// POUs/Local/Objects/FB_BACnet_AV_Disp
// Analog Setpoint Object for Operation
// - Used to display a value
{attribute 'enable_dynamic_creation'}
FUNCTION_BLOCK FB_BACnet_AV_Disp EXTENDS FB_BACnet_Object
VAR_INPUT
	fVal			: REAL;
END_VAR
VAR_INPUT CONSTANT PERSISTENT
	{region 'Variable Parameters'}
		{attribute 'parameterCategory':='Value'}
		fCOVIncrement : REAL := 0.1;
		{attribute 'parameterCategory':='Value'}
		eUnit : E_BA_Unit := E_BA_Unit.eOther_NoUnits;
	{endregion}
END_VAR
VAR_OUTPUT
	fPresVal	: REAL;
END_VAR

IF bReady THEN
	fPresVal := fVal;
ELSE
	fPresVal := 0;
END_IF

SUPER^();

METHOD PROTECTED OnObjectStateChanged
SUPER^.OnObjectStateChanged();

CASE (tState) OF
	TCOM_STATE.TCOM_STATE_PREOP:
		// SyncHandler:
		RequestSyncHandlers(2, 3);
		
		// Properties:
		// EnableProperty(E_BACnetPropIdentifier.PropDeviceType, FALSE);
		EnableProperty(E_BACnetPropIdentifier.PropNotificationClass, FALSE);
		EnableProperty(E_BACnetPropIdentifier.PropNotifyType, FALSE);
		EnableProperty(E_BACnetPropIdentifier.PropEventEnable, FALSE);
		EnableProperty(E_BACnetPropIdentifier.PropEventTimeStamps, FALSE);
		EnableProperty(E_BACnetPropIdentifier.PropEventMessageTexts, FALSE);
		EnableProperty(E_BACnetPropIdentifier.PropEventMessageTextsConfig, FALSE);
		EnableProperty(E_BACnetPropIdentifier.PropTimeDelay, FALSE);
		EnableProperty(E_BACnetPropIdentifier.PropAckedTransitions, FALSE);
		EnableProperty(E_BACnetPropIdentifier.PropReliability, FALSE);
		EnableProperty(E_BACnetPropIdentifier.PropEventDetectionEnable, FALSE);
		EnableProperty(E_BACnetPropIdentifier.PropEventAlgorithmInhibit, FALSE);
		EnableProperty(E_BACnetPropIdentifier.PropTimeDelayNormal, FALSE);
		EnableProperty(E_BACnetPropIdentifier.PropReliabilityEvaluationInhibit, FALSE);
		EnableProperty(E_BACnetPropIdentifier.PropLimitEnable, FALSE);
		EnableProperty(E_BACnetPropIdentifier.PropHighLimit, FALSE);
		EnableProperty(E_BACnetPropIdentifier.PropLowLimit, FALSE);
		EnableProperty(E_BACnetPropIdentifier.PropDeadband, FALSE);
		EnableProperty(E_BACnetPropIdentifier.PropRelinquishDefault, FALSE);
		EnableProperty(E_BACnetPropIdentifier.PropPriorityArray, FALSE);
		EnableProperty(E_BACnetPropIdentifier.PropCurrentlyActivePriority, FALSE);
		
		WriteProtectProperty(E_BACnetPropIdentifier.PropOutOfService, TRUE);
		// EnableProperty(E_BACnetPropIdentifier.PropStatusFlags, FALSE);
		// EnableProperty(E_BACnetPropIdentifier.PropEventState, FALSE);
		
		WriteProtectProperty(E_BACnetPropIdentifier.PropPresentValue, TRUE);

	TCOM_STATE.TCOM_STATE_SAFEOP:
		SyncProperty(E_BACnetPropIdentifier.PropPresentValue, SIZEOF(fVal), ADR(fVal), 0, eSync_ToSupplement);	
	
	TCOM_STATE.TCOM_STATE_OP:
		SyncProperty(E_BACnetPropIdentifier.PropUnits, SIZEOF(eUnit), ADR(eUnit), 0, eFullSync_InitPLC);
		SyncProperty(E_BACnetPropIdentifier.PropCovIncrement, SIZEOF(fCOVIncrement), ADR(fCOVIncrement), 0, eFullSync_InitPLC);
		
END_CASE
END_METHOD

METHOD FB_init : BOOL
VAR_INPUT
	bInitRetains : BOOL; // if TRUE, the retain variables are initialized (warm start / cold start)
	bInCopyCode : BOOL;  // if TRUE, the instance afterwards gets moved into the copy code (online change)
END_VAR
eObjectType := E_BACnetObjType.ObjAnalogValue;
END_METHOD

END_FUNCTION_BLOCK

// POUs/Local/Objects/FB_BACnet_AV_Setp
// Analog Setpoint Object for Operation
// - Used to define a setpoint by user
{attribute 'enable_dynamic_creation'}
FUNCTION_BLOCK FB_BACnet_AV_Setp EXTENDS FB_BACnet_Object
VAR_INPUT CONSTANT PERSISTENT
	{region 'Variable Parameters'}
		{attribute 'parameterCategory':='Value'}
		fCOVIncrement : REAL := 0.1;
		{attribute 'parameterCategory':='Value'}
		eUnit : E_BA_Unit := E_BA_Unit.eOther_NoUnits;
	{endregion}
	{region 'Operational Parameters'}
		{attribute 'parameterCategory':='Value'}
		fValue : REAL;
	{endregion}
END_VAR
VAR_OUTPUT
	fPresVal	: REAL;
END_VAR

IF bReady THEN
	fPresVal := fValue;
ELSE
	fPresVal := 0;
END_IF

SUPER^();

METHOD PROTECTED OnObjectStateChanged
SUPER^.OnObjectStateChanged();

CASE (tState) OF
	TCOM_STATE.TCOM_STATE_PREOP:
		// SyncHandler:
		RequestSyncHandlers(3, 3);
		
		// Properties:
		// DisableProperty(E_BACnetPropIdentifier.PropDeviceType, FALSE);
		EnableProperty(E_BACnetPropIdentifier.PropNotificationClass, FALSE);
		EnableProperty(E_BACnetPropIdentifier.PropNotifyType, FALSE);
		EnableProperty(E_BACnetPropIdentifier.PropEventEnable, FALSE);
		EnableProperty(E_BACnetPropIdentifier.PropEventTimeStamps, FALSE);
		EnableProperty(E_BACnetPropIdentifier.PropEventMessageTexts, FALSE);
		EnableProperty(E_BACnetPropIdentifier.PropEventMessageTextsConfig, FALSE);
		EnableProperty(E_BACnetPropIdentifier.PropTimeDelay, FALSE);
		EnableProperty(E_BACnetPropIdentifier.PropAckedTransitions, FALSE);
		EnableProperty(E_BACnetPropIdentifier.PropReliability, FALSE);
		EnableProperty(E_BACnetPropIdentifier.PropEventDetectionEnable, FALSE);
		EnableProperty(E_BACnetPropIdentifier.PropEventAlgorithmInhibit, FALSE);
		EnableProperty(E_BACnetPropIdentifier.PropTimeDelayNormal, FALSE);
		EnableProperty(E_BACnetPropIdentifier.PropReliabilityEvaluationInhibit, FALSE);
		EnableProperty(E_BACnetPropIdentifier.PropLimitEnable, FALSE);
		EnableProperty(E_BACnetPropIdentifier.PropHighLimit, FALSE);
		EnableProperty(E_BACnetPropIdentifier.PropLowLimit, FALSE);
		EnableProperty(E_BACnetPropIdentifier.PropDeadband, FALSE);
		EnableProperty(E_BACnetPropIdentifier.PropRelinquishDefault, FALSE);
		EnableProperty(E_BACnetPropIdentifier.PropPriorityArray, FALSE);
		EnableProperty(E_BACnetPropIdentifier.PropCurrentlyActivePriority, FALSE);
		
		WriteProtectProperty(E_BACnetPropIdentifier.PropOutOfService, TRUE);
		// EnableProperty(E_BACnetPropIdentifier.PropStatusFlags, FALSE);
		// EnableProperty(E_BACnetPropIdentifier.PropEventState, FALSE);
		
	TCOM_STATE.TCOM_STATE_SAFEOP:
		;
		
	TCOM_STATE.TCOM_STATE_OP:
		SyncProperty(E_BACnetPropIdentifier.PropPresentValue, SIZEOF(fValue), ADR(fValue), 0, eFullSync_InitPLC);
		
		SyncProperty(E_BACnetPropIdentifier.PropUnits, SIZEOF(eUnit), ADR(eUnit), 0, eFullSync_InitPLC);
		SyncProperty(E_BACnetPropIdentifier.PropCovIncrement, SIZEOF(fCOVIncrement), ADR(fCOVIncrement), 0, eFullSync_InitPLC);
		
END_CASE
END_METHOD

METHOD FB_init : BOOL
VAR_INPUT
	bInitRetains : BOOL; // if TRUE, the retain variables are initialized (warm start / cold start)
	bInCopyCode : BOOL;  // if TRUE, the instance afterwards gets moved into the copy code (online change)
END_VAR
eObjectType := E_BACnetObjType.ObjAnalogValue;
END_METHOD

END_FUNCTION_BLOCK

// POUs/Local/Objects/FB_BACnet_BI_Raw
// Binary Input Object
// - Raw communication
{attribute 'pin_presentation_order_outputs' := 'bPresVal,bEvent,eRlbty'}
{attribute 'enable_dynamic_creation'}
FUNCTION_BLOCK FB_BACnet_BI_Raw EXTENDS FB_BACnet_BaseBI
VAR_INPUT
	bRawVal					: BOOL;				// Raw value
END_VAR
VAR_INPUT CONSTANT PERSISTENT
	{region 'Fixed Parameters'}
		{attribute 'parameterCategory':='Hardware'}
		nIoBusNr : BYTE := 16#FF;
	{endregion}
END_VAR

SUPER^();

METHOD PROTECTED OnObjectStateChanged
SUPER^.OnObjectStateChanged();

CASE (tState) OF
	TCOM_STATE.TCOM_STATE_PREOP:
		// SyncHandler:
		RequestSyncHandlers(0, 1);

		IF (nIoBusNr <> 16#FF) THEN
			WritePropertyByte(E_BACnetPropIdentifier.PropIoBusNr, nIoBusNr);
		END_IF
		
	TCOM_STATE.TCOM_STATE_SAFEOP:
		SyncProperty(E_BACnetPropIdentifier.PropRawIoBinaryValueBOOL, SIZEOF(bRawVal), ADR(bRawVal), 0, eSync_ToSupplement);
		
	TCOM_STATE.TCOM_STATE_OP:
		;
		
END_CASE
END_METHOD

END_FUNCTION_BLOCK

// POUs/Local/Objects/[Base]/FB_BACnet_BaseBI
FUNCTION_BLOCK ABSTRACT FB_BACnet_BaseBI EXTENDS FB_BACnet_EventObject
VAR_INPUT CONSTANT PERSISTENT
	{region 'Variable Parameters'}
		{attribute 'parameterCategory':='Value'}
		bOutOfService : BOOL;
		{attribute 'parameterCategory':='Value'}
		{attribute 'TcEncoding':='UTF-8'}
		sInactiveText : T_BACnet_StateText;
		{attribute 'parameterCategory':='Value'}
		{attribute 'TcEncoding':='UTF-8'}
		sActiveText : T_BACnet_StateText;
		
		{attribute 'parameterCategory':='Hardware'}
		{attribute 'TcEncoding':='UTF-8'}
		sDeviceType : STRING;
		
		{attribute 'parameterCategory':='EventConfig'}
		bAlarmValue : BOOL := TRUE;
		
		{attribute 'parameterCategory':='Config'}
		ePolarity : E_BA_Polarity := E_BA_Polarity.eNormal;
			 
		{attribute 'parameterCategory':='StateChange'}
		nChangeOfStateCount : UDINT;
			 
		{attribute 'parameterCategory':='ActiveTime'}
		{attribute 'parameterUnit':= 's'}
		nElapsedActiveTime : UDINT;
	{endregion}
END_VAR
VAR_OUTPUT
	bPresVal			: BOOL;
END_VAR
VAR PERSISTENT 
	{region 'Output-Properties'}
		{attribute 'parameterCategory':='StateChange'}
		stChangeOfStateTime : ST_BA_DateTime;
		{attribute 'parameterCategory':='StateChange'}
		stTimeOfStateCountReset : ST_BA_DateTime;
		
		{attribute 'parameterCategory':='ActiveTime'}
		stTimeOfActiveTimeReset : ST_BA_DateTime;
	{endregion}
END_VAR

SUPER^();

METHOD PROTECTED OnObjectStateChanged
SUPER^.OnObjectStateChanged();

CASE (tState) OF
	TCOM_STATE.TCOM_STATE_PREOP:
		// SyncHandler:
		RequestSyncHandlers(12, 8);
		
		// Properties:
		IF (BACnet_Param.bStateText_WriteProtect) THEN
			WriteProtectProperty(E_BACnetPropIdentifier.PropActiveText, TRUE);
			WriteProtectProperty(E_BACnetPropIdentifier.PropInactiveText, TRUE);
		END_IF
		
		// Ensure UTF-8 Encoding:
		F_BA_EnsureUTF8(ADR(sDeviceType), SIZEOF(sDeviceType));
		F_BA_EnsureUTF8(ADR(sInactiveText), SIZEOF(sInactiveText));
		F_BA_EnsureUTF8(ADR(sActiveText), SIZEOF(sActiveText));

	TCOM_STATE.TCOM_STATE_SAFEOP:
		SyncProperty(E_BACnetPropIdentifier.PropPresentValue, SIZEOF(bPresVal), ADR(bPresVal), 0, eSync_FromSupplement);
		
	TCOM_STATE.TCOM_STATE_OP:
		SyncProperty(E_BACnetPropIdentifier.PropAlarmValue, SIZEOF(bAlarmValue), ADR(bAlarmValue), 0, eFullSync_InitPLC);
		SyncProperty(E_BACnetPropIdentifier.PropOutOfService, SIZEOF(bOutOfService), ADR(bOutOfService), 0, eFullSync_InitPLC);
		SyncProperty(E_BACnetPropIdentifier.PropActiveText, SIZEOF(sActiveText), ADR(sActiveText), 0, eFullSync_InitPLC);	
		SyncProperty(E_BACnetPropIdentifier.PropInactiveText, SIZEOF(sInactiveText), ADR(sInactiveText), 0, eFullSync_InitPLC);
		SyncProperty(E_BACnetPropIdentifier.PropPolarity, SIZEOF(ePolarity), ADR(ePolarity), 0, eFullSync_InitPLC);
		SyncProperty(E_BACnetPropIdentifier.PropDeviceType, SIZEOF(sDeviceType), ADR(sDeviceType), 0, eFullSync_InitPLC);
		SyncProperty(E_BACnetPropIdentifier.PropChangeOfStateCount, SIZEOF(nChangeOfStateCount), ADR(nChangeOfStateCount), 0, eFullSync_InitPLC);
		SyncProperty(E_BACnetPropIdentifier.PropElapsedActiveTime, SIZEOF(nElapsedActiveTime), ADR(nElapsedActiveTime), 0, eFullSync_InitPLC);
		
		SyncProperty(E_BACnetPropIdentifier.PropChangeOfStateTime, SIZEOF(stChangeOfStateTime), ADR(stChangeOfStateTime), 0, eSync_FromSupplementInitPLC);
		SyncProperty(E_BACnetPropIdentifier.PropTimeOfStateCountReset, SIZEOF(stTimeOfStateCountReset), ADR(stTimeOfStateCountReset), 0, eSync_FromSupplementInitPLC);
		SyncProperty(E_BACnetPropIdentifier.PropTimeOfActiveTimeReset, SIZEOF(stTimeOfActiveTimeReset), ADR(stTimeOfActiveTimeReset), 0, eSync_FromSupplementInitPLC);
		
END_CASE
END_METHOD

PROPERTY ChangeOfStateTime : ST_BA_DateTime
GET
ChangeOfStateTime := stChangeOfStateTime;
END_GET
END_PROPERTY

PROPERTY TimeOfActiveTimeReset : ST_BA_DateTime
GET
TimeOfActiveTimeReset := stTimeOfActiveTimeReset;
END_GET
END_PROPERTY

PROPERTY TimeOfStateCountReset : ST_BA_DateTime
GET
TimeOfStateCountReset := stTimeOfStateCountReset;
END_GET
END_PROPERTY

METHOD FB_init : BOOL
VAR_INPUT
	bInitRetains : BOOL; // if TRUE, the retain variables are initialized (warm start / cold start)
	bInCopyCode : BOOL;  // if TRUE, the instance afterwards gets moved into the copy code (online change)
END_VAR
eObjectType := E_BACnetObjType.ObjBinaryInput;
END_METHOD

END_FUNCTION_BLOCK

// POUs/Local/Objects/FB_BACnet_BO_Raw
// Binary Output Object
// - Raw communication
// - 1 Priority
{attribute 'pin_presentation_order_outputs' := 'fPresVal,bEvent,eRlbty'}
{attribute 'enable_dynamic_creation'}
FUNCTION_BLOCK FB_BACnet_BO_Raw EXTENDS FB_BACnet_BaseBO
VAR_INPUT
	bRawOvrrd					: BOOL;				// Raw overridden
	bEnFdbck					: BOOL;				// Enable of writing to Feedback Value (optional)
	bRawValFdbck				: BOOL;				// Raw feedback Value
END_VAR
VAR_OUTPUT
	bRawVal						: BOOL;				// Raw value
END_VAR
VAR_INPUT CONSTANT PERSISTENT
	{region 'Fixed Parameters'}
		{attribute 'parameterCategory':='Hardware'}
		nIoBusNr : BYTE := 16#FF;
	{endregion}
END_VAR

IF (bReady) THEN
	// Feedback Value:
	_bFeedbackValue := SEL(bEnFdbck, bPresVal, bRawValFdbck);
END_IF

SUPER^();

METHOD PROTECTED OnObjectStateChanged
SUPER^.OnObjectStateChanged();

CASE (tState) OF
	TCOM_STATE.TCOM_STATE_PREOP:
		// SyncHandler:
		RequestSyncHandlers(1, 1);

		IF (nIoBusNr <> 16#FF) THEN
			WritePropertyByte(E_BACnetPropIdentifier.PropIoBusNr, nIoBusNr);
		END_IF
		
	TCOM_STATE.TCOM_STATE_SAFEOP:
		SyncProperty(E_BACnetPropIdentifier.PropRawIoBinaryValueBOOL, SIZEOF(bRawVal), ADR(bRawVal), 0, eSync_FromSupplement);
		SyncProperty(E_BACnetPropIdentifier.PropRawIoStateOverride, SIZEOF(bRawOvrrd), ADR(bRawOvrrd), 0, eSync_ToSupplement);
		
	TCOM_STATE.TCOM_STATE_OP:
		;
		
END_CASE
END_METHOD

END_FUNCTION_BLOCK

// POUs/Local/Objects/[Base]/FB_BACnet_BaseBO
FUNCTION_BLOCK ABSTRACT FB_BACnet_BaseBO EXTENDS FB_BACnet_EventObject
VAR_INPUT
	bEnPgm			: BOOL;
	bValPgm			: BOOL;
END_VAR
VAR_INPUT CONSTANT PERSISTENT
	{region 'Variable Parameters'}
		{attribute 'parameterCategory':='General'}
		{attribute 'parameterUnit':= 's'}
		nMinimumOffTime : UDINT;
		{attribute 'parameterCategory':='General'}
		{attribute 'parameterUnit':= 's'}
		nMinimumOnTime : UDINT;
		
		{attribute 'parameterCategory':='Value'}
		bRelinquishDefault : BOOL;
		{attribute 'parameterCategory':='Value'}
		bOutOfService : BOOL;
		{attribute 'parameterCategory':='Value'}
		{attribute 'TcEncoding':='UTF-8'}
		sInactiveText : T_BACnet_StateText;
		{attribute 'parameterCategory':='Value'}
		{attribute 'TcEncoding':='UTF-8'}
		sActiveText : T_BACnet_StateText;
		
		{attribute 'parameterCategory':='Hardware'}
		{attribute 'TcEncoding':='UTF-8'}
		sDeviceType : STRING;
		
		{attribute 'parameterCategory':='Config'}
		ePolarity : E_BA_Polarity := E_BA_Polarity.eNormal;
			 
		{attribute 'parameterCategory':='StateChange'}
		nChangeOfStateCount : UDINT;
			 
		{attribute 'parameterCategory':='ActiveTime'}
		{attribute 'parameterUnit':= 's'}
		nElapsedActiveTime : UDINT;
	{endregion}
END_VAR
VAR_OUTPUT
	bPresVal		: BOOL;
	eActPrio		: E_BACnet_Priority;			// Indicates the currently active priority of the priority array
END_VAR
VAR PERSISTENT
	{region 'Output-Properties'}
		{attribute 'parameterCategory':='StateChange'}
		stChangeOfStateTime : ST_BA_DateTime;
		{attribute 'parameterCategory':='StateChange'}
		stTimeOfStateCountReset : ST_BA_DateTime;
		
		{attribute 'parameterCategory':='ActiveTime'}
		stTimeOfActiveTimeReset : ST_BA_DateTime;
	{endregion}
END_VAR
VAR
	{region 'General'}
		_bFeedbackValue	: BOOL;
	{endregion}
END_VAR

SUPER^();

METHOD PROTECTED OnObjectStateChanged
SUPER^.OnObjectStateChanged();

CASE (tState) OF
	TCOM_STATE.TCOM_STATE_PREOP:
		// SyncHandler:
		RequestSyncHandlers(16, 12);
		
		// Properties:
		IF (BACnet_Param.bStateText_WriteProtect) THEN
			WriteProtectProperty(E_BACnetPropIdentifier.PropActiveText, TRUE);
			WriteProtectProperty(E_BACnetPropIdentifier.PropInactiveText, TRUE);
		END_IF
		
		// Ensure UTF-8 Encoding:
		F_BA_EnsureUTF8(ADR(sDeviceType), SIZEOF(sDeviceType));
		F_BA_EnsureUTF8(ADR(sInactiveText), SIZEOF(sInactiveText));
		F_BA_EnsureUTF8(ADR(sActiveText), SIZEOF(sActiveText));

	TCOM_STATE.TCOM_STATE_SAFEOP:
		SyncPropertyPvPrio(E_BACnetPropIdentifier.PropPresentValue, SIZEOF(bValPgm), ADR(bValPgm), ADR(bEnPgm), BACnet_Param.ePrio_Program, 0, eFullSync_InitPLC);
		
		SyncProperty(E_BACnetPropIdentifier.PropPresentValue, SIZEOF(bPresVal), ADR(bPresVal), 0, eSync_FromSupplement);
		SyncProperty(E_BACnetPropIdentifier.PropCurrentlyActivePriority, SIZEOF(eActPrio), ADR(eActPrio), 0, eSync_FromSupplement);
		
		SyncProperty(E_BACnetPropIdentifier.PropFeedbackValue, SIZEOF(_bFeedbackValue), ADR(_bFeedbackValue), 0, eSync_ToSupplement);
		
	TCOM_STATE.TCOM_STATE_OP:
		SyncProperty(E_BACnetPropIdentifier.PropDeviceType, SIZEOF(sDeviceType), ADR(sDeviceType), 0, eFullSync_InitPLC);
		SyncProperty(E_BACnetPropIdentifier.PropOutOfService, SIZEOF(bOutOfService), ADR(bOutOfService), 0, eFullSync_InitPLC);
		SyncProperty(E_BACnetPropIdentifier.PropMinimumOffTime, SIZEOF(nMinimumOffTime), ADR(nMinimumOffTime), 0, eFullSync_InitPLC);	
		SyncProperty(E_BACnetPropIdentifier.PropMinimumOnTime, SIZEOF(nMinimumOnTime), ADR(nMinimumOnTime), 0, eFullSync_InitPLC);	
		SyncProperty(E_BACnetPropIdentifier.PropRelinquishDefault, SIZEOF(bRelinquishDefault), ADR(bRelinquishDefault), 0, eFullSync_InitPLC);	
		SyncProperty(E_BACnetPropIdentifier.PropActiveText, SIZEOF(sActiveText), ADR(sActiveText), 0, eFullSync_InitPLC);	
		SyncProperty(E_BACnetPropIdentifier.PropInactiveText, SIZEOF(sInactiveText), ADR(sInactiveText), 0, eFullSync_InitPLC);
		SyncProperty(E_BACnetPropIdentifier.PropPolarity, SIZEOF(ePolarity), ADR(ePolarity), 0, eFullSync_InitPLC);
		SyncProperty(E_BACnetPropIdentifier.PropChangeOfStateCount, SIZEOF(nChangeOfStateCount), ADR(nChangeOfStateCount), 0, eFullSync_InitPLC);
		SyncProperty(E_BACnetPropIdentifier.PropElapsedActiveTime, SIZEOF(nElapsedActiveTime), ADR(nElapsedActiveTime), 0, eFullSync_InitPLC);
		
		SyncProperty(E_BACnetPropIdentifier.PropChangeOfStateTime, SIZEOF(stChangeOfStateTime), ADR(stChangeOfStateTime), 0, eSync_FromSupplementInitPLC);
		SyncProperty(E_BACnetPropIdentifier.PropTimeOfStateCountReset, SIZEOF(stTimeOfStateCountReset), ADR(stTimeOfStateCountReset), 0, eSync_FromSupplementInitPLC);
		SyncProperty(E_BACnetPropIdentifier.PropTimeOfActiveTimeReset, SIZEOF(stTimeOfActiveTimeReset), ADR(stTimeOfActiveTimeReset), 0, eSync_FromSupplementInitPLC);
		
END_CASE
END_METHOD

PROPERTY ActivePrio : E_BACnet_Priority
GET
ActivePrio := eActPrio;
END_GET
END_PROPERTY

PROPERTY ChangeOfStateTime : ST_BA_DateTime
GET
ChangeOfStateTime := stChangeOfStateTime;
END_GET
END_PROPERTY

PROPERTY TimeOfActiveTimeReset : ST_BA_DateTime
GET
TimeOfActiveTimeReset := stTimeOfActiveTimeReset;
END_GET
END_PROPERTY

PROPERTY TimeOfStateCountReset : ST_BA_DateTime
GET
TimeOfStateCountReset := stTimeOfStateCountReset;
END_GET
END_PROPERTY

METHOD FB_init : BOOL
VAR_INPUT
	bInitRetains : BOOL; // if TRUE, the retain variables are initialized (warm start / cold start)
	bInCopyCode : BOOL;  // if TRUE, the instance afterwards gets moved into the copy code (online change)
END_VAR
eObjectType := E_BACnetObjType.ObjBinaryOutput;
END_METHOD

END_FUNCTION_BLOCK

// POUs/Local/Objects/[Internal]/5P/FB_BACnet_BO_Raw5P
// Binary Output Object
// - Raw communication
// - 5 Priorities
{attribute 'pin_presentation_order_inputs' := 'bEnSfty,bValSfty,bEnCrit,bValCrit,bEnManLoc,bValManLoc,bEnPgm,bValPgm'}
{attribute 'pin_presentation_order_outputs' := 'bPresVal,eActPrio,bEvent,eRlbty'}
{attribute 'enable_dynamic_creation'}
FUNCTION_BLOCK FB_BACnet_BO_Raw5P EXTENDS FB_BACnet_BO_Raw
VAR_INPUT
	bEnSfty					: BOOL;
	bValSfty				: BOOL;
	bEnCrit					: BOOL;
	bValCrit				: BOOL;
	bEnManLoc				: BOOL;
	bValManLoc				: BOOL;
END_VAR
VAR_INPUT CONSTANT PERSISTENT
	{region 'Operational Parameters'}
		{attribute 'parameterCategory':='Manual'}
		bEnManualOperator : BOOL;
		{attribute 'parameterCategory':='Manual'}
		bValManualOperator : BOOL;
	{endregion}
END_VAR

SUPER^();

METHOD PROTECTED OnObjectStateChanged
SUPER^.OnObjectStateChanged();

CASE (tState) OF
	TCOM_STATE.TCOM_STATE_PREOP:
		// SyncHandler:
		RequestSyncHandlers(4, 4);
		
	TCOM_STATE.TCOM_STATE_SAFEOP:
		SyncPropertyPvPrio(E_BACnetPropIdentifier.PropPresentValue, SIZEOF(bValSfty), ADR(bValSfty), ADR(bEnSfty), BACnet_Param.ePrio_LifeSafety, 0, eFullSync_InitPLC);
		SyncPropertyPvPrio(E_BACnetPropIdentifier.PropPresentValue, SIZEOF(bValCrit), ADR(bValCrit), ADR(bEnCrit), BACnet_Param.ePrio_Critical, 0, eFullSync_InitPLC);
		SyncPropertyPvPrio(E_BACnetPropIdentifier.PropPresentValue, SIZEOF(bValManLoc), ADR(bValManLoc), ADR(bEnManLoc), BACnet_Param.ePrio_ManLocal, 0, eFullSync_InitPLC);
		SyncPropertyPvPrio(E_BACnetPropIdentifier.PropPresentValue, SIZEOF(bValManualOperator), ADR(bValManualOperator), ADR(bEnManualOperator), BACnet_Param.ePrio_ManOperator, 0, eFullSync_InitPLC);
		
	TCOM_STATE.TCOM_STATE_OP:
		;
		
END_CASE
END_METHOD

PROPERTY EnManualOperator : BOOL
GET
EnManualOperator := bEnManualOperator;
END_GET
SET
bEnManualOperator := EnManualOperator;
END_SET
END_PROPERTY

PROPERTY ValManualOperator : BOOL
GET
ValManualOperator := bValManualOperator;
END_GET
SET
bValManualOperator := ValManualOperator;
END_SET
END_PROPERTY

END_FUNCTION_BLOCK

// POUs/Local/Objects/FB_BACnet_BV
// Binary Value Object
// - 1 Priority
{attribute 'enable_dynamic_creation'}
FUNCTION_BLOCK FB_BACnet_BV EXTENDS FB_BACnet_EventObject
VAR_INPUT
	bEnPgm		: BOOL;
	bValPgm		: BOOL;
END_VAR
VAR_INPUT CONSTANT PERSISTENT
	{region 'Variable Parameters'}
		{attribute 'parameterCategory':='General'}
		{attribute 'parameterUnit':= 's'}
		nMinimumOffTime : UDINT;
		{attribute 'parameterCategory':='General'}
		{attribute 'parameterUnit':= 's'}
		nMinimumOnTime : UDINT;
		
		{attribute 'parameterCategory':='Value'}
		bRelinquishDefault : BOOL;
		{attribute 'parameterCategory':='Value'}
		bOutOfService : BOOL;
		{attribute 'parameterCategory':='Value'}
		{attribute 'TcEncoding':='UTF-8'}
		sInactiveText : T_BACnet_StateText;
		{attribute 'parameterCategory':='Value'}
		{attribute 'TcEncoding':='UTF-8'}
		sActiveText : T_BACnet_StateText;
		
		{attribute 'parameterCategory':='EventConfig'}
		bAlarmValue : BOOL := TRUE;
			 
		{attribute 'parameterCategory':='StateChange'}
		nChangeOfStateCount : UDINT;
			 
		{attribute 'parameterCategory':='ActiveTime'}
		{attribute 'parameterUnit':= 's'}
		nElapsedActiveTime : UDINT;
	{endregion}
END_VAR
VAR_OUTPUT
	bPresVal		: BOOL;
	eActPrio		: E_BACnet_Priority;			// Indicates the currently active priority of the priority array
END_VAR
VAR
	{region 'Output-Properties'}
		{attribute 'parameterCategory':='StateChange'}
		stChangeOfStateTime : ST_BA_DateTime;
		{attribute 'parameterCategory':='StateChange'}
		stTimeOfStateCountReset : ST_BA_DateTime;
		
		{attribute 'parameterCategory':='ActiveTime'}
		stTimeOfActiveTimeReset : ST_BA_DateTime;
	{endregion}
END_VAR

SUPER^();

METHOD PROTECTED OnObjectStateChanged
SUPER^.OnObjectStateChanged();

CASE (tState) OF
	TCOM_STATE.TCOM_STATE_PREOP:
		// SyncHandler:
		RequestSyncHandlers(15, 10);
		
		// Properties:
		EnableProperty(E_BACnetPropIdentifier.PropDeviceType, FALSE);

		IF (BACnet_Param.bStateText_WriteProtect) THEN
			WriteProtectProperty(E_BACnetPropIdentifier.PropActiveText, TRUE);
			WriteProtectProperty(E_BACnetPropIdentifier.PropInactiveText, TRUE);
		END_IF
		
		// Ensure UTF-8 Encoding:
		F_BA_EnsureUTF8(ADR(sInactiveText), SIZEOF(sInactiveText));
		F_BA_EnsureUTF8(ADR(sActiveText), SIZEOF(sActiveText));

	TCOM_STATE.TCOM_STATE_SAFEOP:
		SyncPropertyPvPrio(E_BACnetPropIdentifier.PropPresentValue, SIZEOF(bValPgm), ADR(bValPgm), ADR(bEnPgm), BACnet_Param.ePrio_Program, 0, eFullSync_InitPLC);
		
		SyncProperty(E_BACnetPropIdentifier.PropPresentValue, SIZEOF(bPresVal), ADR(bPresVal), 0, eSync_FromSupplement);
		SyncProperty(E_BACnetPropIdentifier.PropCurrentlyActivePriority, SIZEOF(eActPrio), ADR(eActPrio), 0, eSync_FromSupplement);
		
	TCOM_STATE.TCOM_STATE_OP:
		SyncProperty(E_BACnetPropIdentifier.PropAlarmValue, SIZEOF(bAlarmValue), ADR(bAlarmValue), 0, eFullSync_InitPLC);
		SyncProperty(E_BACnetPropIdentifier.PropOutOfService, SIZEOF(bOutOfService), ADR(bOutOfService), 0, eFullSync_InitPLC);
		SyncProperty(E_BACnetPropIdentifier.PropMinimumOffTime, SIZEOF(nMinimumOffTime), ADR(nMinimumOffTime), 0, eFullSync_InitPLC);	
		SyncProperty(E_BACnetPropIdentifier.PropMinimumOnTime, SIZEOF(nMinimumOnTime), ADR(nMinimumOnTime), 0, eFullSync_InitPLC);	
		SyncProperty(E_BACnetPropIdentifier.PropRelinquishDefault, SIZEOF(bRelinquishDefault), ADR(bRelinquishDefault), 0, eFullSync_InitPLC);	
		SyncProperty(E_BACnetPropIdentifier.PropActiveText, SIZEOF(sActiveText), ADR(sActiveText), 0, eFullSync_InitPLC);	
		SyncProperty(E_BACnetPropIdentifier.PropInactiveText, SIZEOF(sInactiveText), ADR(sInactiveText), 0, eFullSync_InitPLC);
		SyncProperty(E_BACnetPropIdentifier.PropChangeOfStateCount, SIZEOF(nChangeOfStateCount), ADR(nChangeOfStateCount), 0, eFullSync_InitPLC);
		SyncProperty(E_BACnetPropIdentifier.PropElapsedActiveTime, SIZEOF(nElapsedActiveTime), ADR(nElapsedActiveTime), 0, eFullSync_InitPLC);
		
		SyncProperty(E_BACnetPropIdentifier.PropChangeOfStateTime, SIZEOF(stChangeOfStateTime), ADR(stChangeOfStateTime), 0, eSync_FromSupplementInitPLC);
		SyncProperty(E_BACnetPropIdentifier.PropTimeOfStateCountReset, SIZEOF(stTimeOfStateCountReset), ADR(stTimeOfStateCountReset), 0, eSync_FromSupplementInitPLC);
		SyncProperty(E_BACnetPropIdentifier.PropTimeOfActiveTimeReset, SIZEOF(stTimeOfActiveTimeReset), ADR(stTimeOfActiveTimeReset), 0, eSync_FromSupplementInitPLC);
		
END_CASE
END_METHOD

PROPERTY ActivePrio : E_BACnet_Priority
GET
ActivePrio := eActPrio;
END_GET
END_PROPERTY

PROPERTY ChangeOfStateTime : ST_BA_DateTime
GET
ChangeOfStateTime := stChangeOfStateTime;
END_GET
END_PROPERTY

PROPERTY TimeOfActiveTimeReset : ST_BA_DateTime
GET
TimeOfActiveTimeReset := stTimeOfActiveTimeReset;
END_GET
END_PROPERTY

PROPERTY TimeOfStateCountReset : ST_BA_DateTime
GET
TimeOfStateCountReset := stTimeOfStateCountReset;
END_GET
END_PROPERTY

METHOD FB_init : BOOL
VAR_INPUT
	bInitRetains : BOOL; // if TRUE, the retain variables are initialized (warm start / cold start)
	bInCopyCode : BOOL;  // if TRUE, the instance afterwards gets moved into the copy code (online change)
END_VAR
eObjectType := E_BACnetObjType.ObjBinaryValue;
END_METHOD

END_FUNCTION_BLOCK

// POUs/Local/Objects/[Internal]/5P/FB_BACnet_BV_5P
// Binary Value Object
// - 5 Priorities
{attribute 'pin_presentation_order_inputs' := 'bEnSfty,bValSfty,bEnCrit,bValCrit,bEnManLoc,bValManLoc,bEnPgm,bValPgm'}
{attribute 'pin_presentation_order_outputs' := 'bPresVal,eActPrio,bEvent,eRlbty'}
{attribute 'enable_dynamic_creation'}
FUNCTION_BLOCK FB_BACnet_BV_5P EXTENDS FB_BACnet_BV
VAR_INPUT
	bEnSfty					: BOOL;
	bValSfty				: BOOL;
	bEnCrit					: BOOL;
	bValCrit				: BOOL;
	bEnManLoc				: BOOL;
	bValManLoc				: BOOL;
END_VAR
VAR_INPUT CONSTANT PERSISTENT
	{region 'Operational Parameters'}
		{attribute 'parameterCategory':='Manual'}
		bEnManualOperator : BOOL;
		{attribute 'parameterCategory':='Manual'}
		bValManualOperator : BOOL;
	{endregion}
END_VAR

SUPER^();

METHOD PROTECTED OnObjectStateChanged
SUPER^.OnObjectStateChanged();

CASE (tState) OF
	TCOM_STATE.TCOM_STATE_PREOP:
		// SyncHandler:
		RequestSyncHandlers(4, 4);
		
	TCOM_STATE.TCOM_STATE_SAFEOP:
		SyncPropertyPvPrio(E_BACnetPropIdentifier.PropPresentValue, SIZEOF(bValSfty), ADR(bValSfty), ADR(bEnSfty), BACnet_Param.ePrio_LifeSafety, 0, eFullSync_InitPLC);
		SyncPropertyPvPrio(E_BACnetPropIdentifier.PropPresentValue, SIZEOF(bValCrit), ADR(bValCrit), ADR(bEnCrit), BACnet_Param.ePrio_Critical, 0, eFullSync_InitPLC);
		SyncPropertyPvPrio(E_BACnetPropIdentifier.PropPresentValue, SIZEOF(bValManLoc), ADR(bValManLoc), ADR(bEnManLoc), BACnet_Param.ePrio_ManLocal, 0, eFullSync_InitPLC);
		SyncPropertyPvPrio(E_BACnetPropIdentifier.PropPresentValue, SIZEOF(bValManualOperator), ADR(bValManualOperator), ADR(bEnManualOperator), BACnet_Param.ePrio_ManOperator, 0, eFullSync_InitPLC);
		
	TCOM_STATE.TCOM_STATE_OP:
		;
		
END_CASE
END_METHOD

PROPERTY EnManualOperator : BOOL
GET
EnManualOperator := bEnManualOperator;
END_GET
SET
bEnManualOperator := EnManualOperator;
END_SET
END_PROPERTY

PROPERTY ValManualOperator : BOOL
GET
ValManualOperator := bValManualOperator;
END_GET
SET
bValManualOperator := ValManualOperator;
END_SET
END_PROPERTY

END_FUNCTION_BLOCK

// POUs/Local/Objects/FB_BACnet_BV_Disp
// Binary Setpoint Object for Operation
// - Used to display a value
{attribute 'enable_dynamic_creation'}
FUNCTION_BLOCK FB_BACnet_BV_Disp EXTENDS FB_BACnet_Object
VAR_INPUT
	bVal			: BOOL;
END_VAR
VAR_INPUT CONSTANT PERSISTENT
	{region 'Variable Parameters'}
		{attribute 'parameterCategory':='Value'}
		{attribute 'TcEncoding':='UTF-8'}
		sInactiveText : T_BACnet_StateText;
		{attribute 'parameterCategory':='Value'}
		{attribute 'TcEncoding':='UTF-8'}
		sActiveText : T_BACnet_StateText;
	{endregion}
END_VAR
VAR_OUTPUT
	bPresVal	: BOOL;
END_VAR

IF bReady THEN
	bPresVal := bVal;
ELSE
	bPresVal := FALSE;
END_IF

SUPER^();

METHOD PROTECTED OnObjectStateChanged
SUPER^.OnObjectStateChanged();

CASE (tState) OF
	TCOM_STATE.TCOM_STATE_PREOP:
		// SyncHandler:
		RequestSyncHandlers(2, 3);
		
		// Properties:
		EnableProperty(E_BACnetPropIdentifier.PropDeviceType, FALSE);
		EnableProperty(E_BACnetPropIdentifier.PropMinimumOnTime, FALSE);
		EnableProperty(E_BACnetPropIdentifier.PropMinimumOffTime, FALSE);
		EnableProperty(E_BACnetPropIdentifier.PropNotificationClass, FALSE);
		EnableProperty(E_BACnetPropIdentifier.PropNotifyType, FALSE);
		EnableProperty(E_BACnetPropIdentifier.PropEventEnable, FALSE);
		EnableProperty(E_BACnetPropIdentifier.PropEventTimeStamps, FALSE);
		EnableProperty(E_BACnetPropIdentifier.PropEventMessageTexts, FALSE);
		EnableProperty(E_BACnetPropIdentifier.PropEventMessageTextsConfig, FALSE);
		EnableProperty(E_BACnetPropIdentifier.PropTimeDelay, FALSE);
		EnableProperty(E_BACnetPropIdentifier.PropAckedTransitions, FALSE);
		EnableProperty(E_BACnetPropIdentifier.PropReliability, FALSE);
		EnableProperty(E_BACnetPropIdentifier.PropEventDetectionEnable, FALSE);
		EnableProperty(E_BACnetPropIdentifier.PropEventAlgorithmInhibit, FALSE);
		EnableProperty(E_BACnetPropIdentifier.PropTimeDelayNormal, FALSE);
		EnableProperty(E_BACnetPropIdentifier.PropReliabilityEvaluationInhibit, FALSE);
		EnableProperty(E_BACnetPropIdentifier.PropChangeOfStateCount, FALSE);
		EnableProperty(E_BACnetPropIdentifier.PropChangeOfStateTime, FALSE);
		EnableProperty(E_BACnetPropIdentifier.PropTimeOfStateCountReset, FALSE);
		EnableProperty(E_BACnetPropIdentifier.PropElapsedActiveTime, FALSE);
		EnableProperty(E_BACnetPropIdentifier.PropTimeOfActiveTimeReset, FALSE);
		EnableProperty(E_BACnetPropIdentifier.PropRelinquishDefault, FALSE);
		EnableProperty(E_BACnetPropIdentifier.PropPriorityArray, FALSE);
		EnableProperty(E_BACnetPropIdentifier.PropCurrentlyActivePriority, FALSE);
		
		WriteProtectProperty(E_BACnetPropIdentifier.PropOutOfService, TRUE);
		// EnableProperty(E_BACnetPropIdentifier.PropStatusFlags, FALSE);
		// EnableProperty(E_BACnetPropIdentifier.PropEventState, FALSE);
		
		WriteProtectProperty(E_BACnetPropIdentifier.PropPresentValue, TRUE);
		
		IF (BACnet_Param.bStateText_WriteProtect) THEN
			WriteProtectProperty(E_BACnetPropIdentifier.PropActiveText, TRUE);
			WriteProtectProperty(E_BACnetPropIdentifier.PropInactiveText, TRUE);
		END_IF
		
		// Ensure UTF-8 Encoding:
		F_BA_EnsureUTF8(ADR(sInactiveText), SIZEOF(sInactiveText));
		F_BA_EnsureUTF8(ADR(sActiveText), SIZEOF(sActiveText));
		
	TCOM_STATE.TCOM_STATE_SAFEOP:
		SyncProperty(E_BACnetPropIdentifier.PropPresentValue, SIZEOF(bVal), ADR(bVal), 0, eSync_ToSupplement);
		
	TCOM_STATE.TCOM_STATE_OP:
		SyncProperty(E_BACnetPropIdentifier.PropActiveText, SIZEOF(sActiveText), ADR(sActiveText), 0, eFullSync_InitPLC);	
		SyncProperty(E_BACnetPropIdentifier.PropInactiveText, SIZEOF(sInactiveText), ADR(sInactiveText), 0, eFullSync_InitPLC);
		
END_CASE
END_METHOD

METHOD FB_init : BOOL
VAR_INPUT
	bInitRetains : BOOL; // if TRUE, the retain variables are initialized (warm start / cold start)
	bInCopyCode : BOOL;  // if TRUE, the instance afterwards gets moved into the copy code (online change)
END_VAR
eObjectType := E_BACnetObjType.ObjBinaryValue;
END_METHOD

END_FUNCTION_BLOCK

// POUs/Local/Objects/FB_BACnet_BV_Setp
// Binary Setpoint Object for Operation
// - Used to define a setpoint by user
{attribute 'enable_dynamic_creation'}
FUNCTION_BLOCK FB_BACnet_BV_Setp EXTENDS FB_BACnet_Object
VAR_INPUT CONSTANT PERSISTENT
	{region 'Variable Parameters'}
		{attribute 'parameterCategory':='Value'}
		{attribute 'TcEncoding':='UTF-8'}
		sInactiveText : T_BACnet_StateText;
		{attribute 'parameterCategory':='Value'}
		{attribute 'TcEncoding':='UTF-8'}
		sActiveText : T_BACnet_StateText;
	{endregion}
	{region 'Operational Parameters'}
		{attribute 'parameterCategory':='Value'}
		bValue : BOOL;
	{endregion}
END_VAR
VAR_OUTPUT
	bPresVal	: BOOL;
END_VAR

IF bReady THEN
	bPresVal := bValue;
ELSE
	bPresVal := FALSE;
END_IF

SUPER^();

METHOD PROTECTED OnObjectStateChanged
SUPER^.OnObjectStateChanged();

CASE (tState) OF
	TCOM_STATE.TCOM_STATE_PREOP:
		// SyncHandler:
		RequestSyncHandlers(3, 3);
		
		// Properties:
		EnableProperty(E_BACnetPropIdentifier.PropDeviceType, FALSE);
		EnableProperty(E_BACnetPropIdentifier.PropMinimumOnTime, FALSE);
		EnableProperty(E_BACnetPropIdentifier.PropMinimumOffTime, FALSE);
		EnableProperty(E_BACnetPropIdentifier.PropNotificationClass, FALSE);
		EnableProperty(E_BACnetPropIdentifier.PropNotifyType, FALSE);
		EnableProperty(E_BACnetPropIdentifier.PropEventEnable, FALSE);
		EnableProperty(E_BACnetPropIdentifier.PropEventTimeStamps, FALSE);
		EnableProperty(E_BACnetPropIdentifier.PropEventMessageTexts, FALSE);
		EnableProperty(E_BACnetPropIdentifier.PropEventMessageTextsConfig, FALSE);
		EnableProperty(E_BACnetPropIdentifier.PropTimeDelay, FALSE);
		EnableProperty(E_BACnetPropIdentifier.PropAckedTransitions, FALSE);
		EnableProperty(E_BACnetPropIdentifier.PropReliability, FALSE);
		EnableProperty(E_BACnetPropIdentifier.PropEventDetectionEnable, FALSE);
		EnableProperty(E_BACnetPropIdentifier.PropEventAlgorithmInhibit, FALSE);
		EnableProperty(E_BACnetPropIdentifier.PropTimeDelayNormal, FALSE);
		EnableProperty(E_BACnetPropIdentifier.PropReliabilityEvaluationInhibit, FALSE);
		EnableProperty(E_BACnetPropIdentifier.PropChangeOfStateCount, FALSE);
		EnableProperty(E_BACnetPropIdentifier.PropChangeOfStateTime, FALSE);
		EnableProperty(E_BACnetPropIdentifier.PropTimeOfStateCountReset, FALSE);
		EnableProperty(E_BACnetPropIdentifier.PropElapsedActiveTime, FALSE);
		EnableProperty(E_BACnetPropIdentifier.PropTimeOfActiveTimeReset, FALSE);
		EnableProperty(E_BACnetPropIdentifier.PropRelinquishDefault, FALSE);
		EnableProperty(E_BACnetPropIdentifier.PropPriorityArray, FALSE);
		EnableProperty(E_BACnetPropIdentifier.PropCurrentlyActivePriority, FALSE);
		
		WriteProtectProperty(E_BACnetPropIdentifier.PropOutOfService, TRUE);
		// EnableProperty(E_BACnetPropIdentifier.PropStatusFlags, FALSE);
		// EnableProperty(E_BACnetPropIdentifier.PropEventState, FALSE);
		
		IF (BACnet_Param.bStateText_WriteProtect) THEN
			WriteProtectProperty(E_BACnetPropIdentifier.PropActiveText, TRUE);
			WriteProtectProperty(E_BACnetPropIdentifier.PropInactiveText, TRUE);
		END_IF
		
		// Ensure UTF-8 Encoding:
		F_BA_EnsureUTF8(ADR(sInactiveText), SIZEOF(sInactiveText));
		F_BA_EnsureUTF8(ADR(sActiveText), SIZEOF(sActiveText));
		
	TCOM_STATE.TCOM_STATE_SAFEOP:
		;
		
	TCOM_STATE.TCOM_STATE_OP:
		SyncProperty(E_BACnetPropIdentifier.PropPresentValue, SIZEOF(bValue), ADR(bValue), 0, eFullSync_InitPLC);
		
		SyncProperty(E_BACnetPropIdentifier.PropActiveText, SIZEOF(sActiveText), ADR(sActiveText), 0, eFullSync_InitPLC);	
		SyncProperty(E_BACnetPropIdentifier.PropInactiveText, SIZEOF(sInactiveText), ADR(sInactiveText), 0, eFullSync_InitPLC);
		
END_CASE
END_METHOD

METHOD FB_init : BOOL
VAR_INPUT
	bInitRetains : BOOL; // if TRUE, the retain variables are initialized (warm start / cold start)
	bInCopyCode : BOOL;  // if TRUE, the instance afterwards gets moved into the copy code (online change)
END_VAR
eObjectType := E_BACnetObjType.ObjBinaryValue;
END_METHOD

END_FUNCTION_BLOCK

// POUs/Local/Objects/FB_BACnet_MI_Raw
// Multistate Input Object
// - Raw communication
{attribute 'pin_presentation_order_outputs' := 'nPresVal,bEvent,eRlbty'}
{attribute 'enable_dynamic_creation'}
FUNCTION_BLOCK FB_BACnet_MI_Raw EXTENDS FB_BACnet_BaseMI
VAR_INPUT
	nRawValue		: UDINT		:= 1;			// Raw value
END_VAR

SUPER^();

METHOD PROTECTED OnObjectStateChanged
SUPER^.OnObjectStateChanged();

CASE (tState) OF
	TCOM_STATE.TCOM_STATE_PREOP:
		// SyncHandler:
		RequestSyncHandlers(0, 1);
		
	TCOM_STATE.TCOM_STATE_SAFEOP:
		SyncProperty(E_BACnetPropIdentifier.PropPresentValue, SIZEOF(nRawValue), ADR(nRawValue), 0, eSync_ToSupplement);
		
	TCOM_STATE.TCOM_STATE_OP:
		;
		
END_CASE
END_METHOD

END_FUNCTION_BLOCK

// POUs/Local/Objects/[Base]/FB_BACnet_BaseMI
FUNCTION_BLOCK ABSTRACT FB_BACnet_BaseMI EXTENDS FB_BACnet_EventObject
VAR_INPUT CONSTANT PERSISTENT
	{region 'Variable Parameters'}
		{attribute 'parameterCategory':='Value'}
		bOutOfService : BOOL;
		
		{attribute 'parameterCategory':='Hardware'}
		{attribute 'TcEncoding':='UTF-8'}
		sDeviceType : STRING;
	{endregion}
	{region 'Fixed Parameters'}
		{attribute 'parameterCategory':='Value'}
		{attribute 'TcEncoding':='UTF-8'}
		aStateText : T_BACnet_StateTextArray := BACnet_Param.sMultistate_DefaultStateText;
		
		{attribute 'parameterCategory':='EventConfig'}
		aAlarmValues : T_BACnet_MultistateValue;
		{attribute 'parameterCategory':='EventConfig'}
		aFaultValues : T_BACnet_MultistateValue;
	{endregion}
END_VAR
VAR_OUTPUT
	nPresVal			: UDINT		:= 1;
END_VAR
VAR
	{region 'Output-Properties'}
		nStateCount		: UDINT;
	{endregion}
END_VAR

SUPER^();

METHOD PROTECTED OnObjectStateChanged
SUPER^.OnObjectStateChanged();

CASE (tState) OF
	TCOM_STATE.TCOM_STATE_PREOP:
		{warning disable C0196}
		nStateCount := F_BACnet_GetUsedStateText(aStateText);
		
		// SyncHandler:
		RequestSyncHandlers(nStateCount, nStateCount);						// Handlers for "E_BACnetPropIdentifier.PropStateText"
		_nTemp := F_BACnet_GetUsedUDINT(aAlarmValues);						// Handlers for "E_BACnetPropIdentifier.PropAlarmValues"
		RequestSyncHandlers(_nTemp, _nTemp);
		_nTemp := F_BACnet_GetUsedUDINT(aFaultValues);						// Handlers for "E_BACnetPropIdentifier.PropFaultValues"
		RequestSyncHandlers(_nTemp, _nTemp);
		RequestSyncHandlers(5, 6);											// Handlers for other properties
		{warning restore C0196}
		
		// Properties:
		WriteProtectProperty(E_BACnetPropIdentifier.PropNumberOfStates, TRUE);
		
		IF (BACnet_Param.bStateText_WriteProtect) THEN
			WriteProtectProperty(E_BACnetPropIdentifier.PropStateText, TRUE);
		END_IF
		
		// Ensure UTF-8 Encoding:
		F_BA_EnsureUTF8(ADR(sDeviceType), SIZEOF(sDeviceType));
		F_BA_EnsureUTF8Array(ADR(aStateText), SIZEOF(aStateText[1]), TO_DINT(BACnet_Param.nMultistate_StateCount));

	TCOM_STATE.TCOM_STATE_SAFEOP:
		SyncProperty(E_BACnetPropIdentifier.PropPresentValue, SIZEOF(nPresVal), ADR(nPresVal), 0, eSync_FromSupplement);
			
	TCOM_STATE.TCOM_STATE_OP:
		// Init number of used states:
		SetNumberOfStates(nStateCount);
		
		SyncProperty(E_BACnetPropIdentifier.PropOutOfService, SIZEOF(bOutOfService), ADR(bOutOfService), 0, eFullSync_InitPLC);
		SyncProperty(E_BACnetPropIdentifier.PropDeviceType, SIZEOF(sDeviceType), ADR(sDeviceType), 0, eFullSync_InitPLC);
		SyncPropertyList(E_BACnetPropIdentifier.PropStateText, ADR(aStateText), SIZEOF(T_BACnet_StateText), nStateCount, eFullSync_InitPLC, FALSE);
		SyncPropertyList(E_BACnetPropIdentifier.PropAlarmValues, ADR(aAlarmValues), SIZEOF(UDINT), nStateCount, eFullSync_InitPLC, TRUE);
		SyncPropertyList(E_BACnetPropIdentifier.PropFaultValues, ADR(aFaultValues), SIZEOF(UDINT), nStateCount, eFullSync_InitPLC, TRUE);

END_CASE
END_METHOD

PROPERTY StateCount : UDINT
GET
StateCount := nStateCount;
END_GET
END_PROPERTY

METHOD FB_init : BOOL
VAR_INPUT
	bInitRetains : BOOL; // if TRUE, the retain variables are initialized (warm start / cold start)
	bInCopyCode : BOOL;  // if TRUE, the instance afterwards gets moved into the copy code (online change)
END_VAR
eObjectType := E_BACnetObjType.ObjMultistateInput;
END_METHOD

END_FUNCTION_BLOCK

// POUs/Helper/[internal]/String/F_BACnet_GetUsedStateText
{attribute 'hide'}
FUNCTION F_BACnet_GetUsedStateText : UDINT
VAR_IN_OUT
	aArray				: ARRAY[*] OF T_BACnet_StateText;
END_VAR
VAR
	_nTemp				: DINT;
END_VAR

F_BACnet_GetUsedStateText := 0;

FOR _nTemp := LOWER_BOUND(aArray, 1) TO UPPER_BOUND(aArray, 1) DO
	IF LEN(aArray[_nTemp]) = 0 THEN
		EXIT;
	ELSE
		F_BACnet_GetUsedStateText := (F_BACnet_GetUsedStateText+1);
	END_IF
END_FOR

END_FUNCTION

// POUs/Helper/[internal]/String/F_BACnet_GetUsedUDINT
{attribute 'hide'}
FUNCTION F_BACnet_GetUsedUDINT : UDINT
VAR_IN_OUT
	aArray				: ARRAY[*] OF UDINT;
END_VAR
VAR
	_nTemp				: DINT;
END_VAR

F_BACnet_GetUsedUDINT := 0;

FOR _nTemp := LOWER_BOUND(aArray, 1) TO UPPER_BOUND(aArray, 1) DO
	IF (aArray[_nTemp] = 0) THEN
		EXIT;
	ELSE
		F_BACnet_GetUsedUDINT := (F_BACnet_GetUsedUDINT+1);
	END_IF
END_FOR

END_FUNCTION

// POUs/Local/Objects/FB_BACnet_MO_Raw
// Multistate Output Object
// - Raw communication
// - 1 Priority
{attribute 'pin_presentation_order_outputs' := 'fPresVal,bEvent,eRlbty'}
{attribute 'enable_dynamic_creation'}
FUNCTION_BLOCK FB_BACnet_MO_Raw EXTENDS FB_BACnet_BaseMO
VAR_INPUT
	bRawOvrrd					: BOOL;				// Raw overridden
	bEnFeedback					: BOOL;				// Enable of writing to Feedback Value (optional)
	nRawValFeedback				: UDINT;			// Raw feedback Value
END_VAR
VAR_OUTPUT
	nRawValue					: UDINT;			// Raw value
END_VAR

IF (bReady) THEN
	// Feedback Value:
	_nFeedbackValue := MAX(1, SEL(bEnFeedback, nPresVal, nRawValFeedback));
	
	// Raw-IO Value:
	nRawValue := nPresVal;
END_IF

SUPER^();

METHOD PROTECTED OnObjectStateChanged
SUPER^.OnObjectStateChanged();

CASE (tState) OF
	TCOM_STATE.TCOM_STATE_PREOP:
		// SyncHandler:
		RequestSyncHandlers(0, 1);

	TCOM_STATE.TCOM_STATE_SAFEOP:
		SyncProperty(E_BACnetPropIdentifier.PropRawIoStateOverride, SIZEOF(bRawOvrrd), ADR(bRawOvrrd), 0, eSync_ToSupplement);
		
	TCOM_STATE.TCOM_STATE_OP:
		;

END_CASE
END_METHOD

END_FUNCTION_BLOCK

// POUs/Local/Objects/[Base]/FB_BACnet_BaseMO
FUNCTION_BLOCK ABSTRACT FB_BACnet_BaseMO EXTENDS FB_BACnet_EventObject
VAR_INPUT
	bEnPgm					: BOOL;
	nValPgm					: UDINT		:= 1;
END_VAR
VAR_INPUT CONSTANT PERSISTENT
	{region 'Variable Parameters'}
		{attribute 'parameterCategory':='Value'}
		nRelinquishDefault : UDINT := 1;
		{attribute 'parameterCategory':='Value'}
		bOutOfService : BOOL;
	
		{attribute 'parameterCategory':='Hardware'}
		{attribute 'TcEncoding':='UTF-8'}
		sDeviceType : STRING;
	{endregion}
	{region 'Fixed Parameters'}
		{attribute 'parameterCategory':='Value'}
		{attribute 'TcEncoding':='UTF-8'}
		sStateText : T_BACnet_StateTextArray := BACnet_Param.sMultistate_DefaultStateText;
	{endregion}
END_VAR
VAR_OUTPUT
	nPresVal				: UDINT		:= 1;
	eActPrio				: E_BACnet_Priority;			// Indicates the currently active priority of the priority array
END_VAR
VAR
	{region 'Output-Properties'}
		nStateCount			: UDINT;
	{endregion}
END_VAR
VAR
	{region 'Internal'}
		_nFeedbackValue		: UDINT;
	{endregion}
END_VAR

SUPER^();

METHOD PROTECTED OnObjectStateChanged
SUPER^.OnObjectStateChanged();

CASE (tState) OF
	TCOM_STATE.TCOM_STATE_PREOP:
		// SyncHandler:
		{warning disable C0196}
		nStateCount := F_BACnet_GetUsedStateText(sStateText);
		{warning restore C0196}
		
		RequestSyncHandlers(nStateCount, nStateCount);						// Handlers for "E_BACnetPropIdentifier.PropStateText"
		RequestSyncHandlers(7, 6);											// Handlers for other properties
		
		// Properties:
		WriteProtectProperty(E_BACnetPropIdentifier.PropNumberOfStates, TRUE);
		
		IF (BACnet_Param.bStateText_WriteProtect) THEN
			WriteProtectProperty(E_BACnetPropIdentifier.PropStateText, TRUE);
		END_IF
		
		// Ensure UTF-8 Encoding:
		F_BA_EnsureUTF8(ADR(sDeviceType), SIZEOF(sDeviceType));
		F_BA_EnsureUTF8Array(ADR(sStateText), SIZEOF(sStateText[1]), TO_DINT(BACnet_Param.nMultistate_StateCount));
		
	TCOM_STATE.TCOM_STATE_SAFEOP:
		SyncPropertyPvPrio(E_BACnetPropIdentifier.PropPresentValue, SIZEOF(nValPgm), ADR(nValPgm), ADR(bEnPgm), BACnet_Param.ePrio_Program, 0, eFullSync_InitPLC);
		
		SyncProperty(E_BACnetPropIdentifier.PropPresentValue, SIZEOF(nPresVal), ADR(nPresVal), 0, eSync_FromSupplement);
		SyncProperty(E_BACnetPropIdentifier.PropCurrentlyActivePriority, SIZEOF(eActPrio), ADR(eActPrio), 0, eSync_FromSupplement);
		
		SyncProperty(E_BACnetPropIdentifier.PropFeedbackValue, SIZEOF(_nFeedbackValue), ADR(_nFeedbackValue), 0, eSync_ToSupplement);
		
	TCOM_STATE.TCOM_STATE_OP:
		// Init number of used states:
		SetNumberOfStates(nStateCount);
		
		SyncProperty(E_BACnetPropIdentifier.PropDeviceType, SIZEOF(sDeviceType), ADR(sDeviceType), 0, eFullSync_InitPLC);
		SyncProperty(E_BACnetPropIdentifier.PropRelinquishDefault, SIZEOF(nRelinquishDefault), ADR(nRelinquishDefault), 0, eFullSync_InitPLC);
		SyncProperty(E_BACnetPropIdentifier.PropOutOfService, SIZEOF(bOutOfService), ADR(bOutOfService), 0, eFullSync_InitPLC);
		SyncPropertyList(E_BACnetPropIdentifier.PropStateText, ADR(sStateText), SIZEOF(T_BACnet_StateText), nStateCount, eFullSync_InitPLC, FALSE);
		
END_CASE
END_METHOD

PROPERTY ActivePrio : E_BACnet_Priority
GET
ActivePrio := eActPrio;
END_GET
END_PROPERTY

PROPERTY StateCount : UDINT
GET
StateCount := nStateCount;
END_GET
END_PROPERTY

METHOD FB_init : BOOL
VAR_INPUT
	bInitRetains : BOOL; // if TRUE, the retain variables are initialized (warm start / cold start)
	bInCopyCode : BOOL;  // if TRUE, the instance afterwards gets moved into the copy code (online change)
END_VAR
eObjectType := E_BACnetObjType.ObjMultistateOutput;
END_METHOD

END_FUNCTION_BLOCK

// POUs/Local/Objects/[Internal]/5P/FB_BACnet_MO_Raw5P
// Multistate Output Object
// - Raw communication
// - 5 Priorities
{attribute 'pin_presentation_order_inputs' := 'bEnSfty,nValSfty,bEnCrit,nValCrit,bEnManLoc,nValManLoc,bEnPgm,nValPgm'}
{attribute 'pin_presentation_order_outputs' := 'nPresVal,eActPrio,bEvent,eRlbty'}
{attribute 'enable_dynamic_creation'}
FUNCTION_BLOCK FB_BACnet_MO_Raw5P EXTENDS FB_BACnet_MO_Raw
VAR_INPUT
	bEnSfty					: BOOL;
	nValSfty				: UDINT		:= 1;
	bEnCrit					: BOOL;
	nValCrit				: UDINT		:= 1;
	bEnManLoc				: BOOL;
	nValManLoc				: UDINT		:= 1;
END_VAR
VAR_INPUT CONSTANT PERSISTENT
	{region 'Operational Parameters'}
		{attribute 'parameterCategory':='Manual'}
		bEnManualOperator : BOOL;
		{attribute 'parameterCategory':='Manual'}
		nValManualOperator : UDINT := 1;
	{endregion}
END_VAR

SUPER^();

METHOD PROTECTED OnObjectStateChanged
SUPER^.OnObjectStateChanged();

CASE (tState) OF
	TCOM_STATE.TCOM_STATE_PREOP:
		// SyncHandler:
		RequestSyncHandlers(4, 4);
		
	TCOM_STATE.TCOM_STATE_SAFEOP:
		SyncPropertyPvPrio(E_BACnetPropIdentifier.PropPresentValue, SIZEOF(nValSfty), ADR(nValSfty), ADR(bEnSfty), BACnet_Param.ePrio_LifeSafety, 0, eFullSync_InitPLC);
		SyncPropertyPvPrio(E_BACnetPropIdentifier.PropPresentValue, SIZEOF(nValCrit), ADR(nValCrit), ADR(bEnCrit), BACnet_Param.ePrio_Critical, 0, eFullSync_InitPLC);
		SyncPropertyPvPrio(E_BACnetPropIdentifier.PropPresentValue, SIZEOF(nValManLoc), ADR(nValManLoc), ADR(bEnManLoc), BACnet_Param.ePrio_ManLocal, 0, eFullSync_InitPLC);
		SyncPropertyPvPrio(E_BACnetPropIdentifier.PropPresentValue, SIZEOF(nValManualOperator), ADR(nValManualOperator), ADR(bEnManualOperator), BACnet_Param.ePrio_ManOperator, 0, eFullSync_InitPLC);
		
	TCOM_STATE.TCOM_STATE_OP:
		;
		
END_CASE
END_METHOD

PROPERTY EnManualOperator : BOOL
GET
EnManualOperator := bEnManualOperator;
END_GET
SET
bEnManualOperator := EnManualOperator;
END_SET
END_PROPERTY

PROPERTY ValManualOperator : UDINT
GET
ValManualOperator := nValManualOperator;
END_GET
SET
nValManualOperator := ValManualOperator;
END_SET
END_PROPERTY

END_FUNCTION_BLOCK

// POUs/Local/Objects/FB_BACnet_MV
// Multistate Value Object
// - 1 Priority
{attribute 'enable_dynamic_creation'}
FUNCTION_BLOCK FB_BACnet_MV EXTENDS FB_BACnet_EventObject
VAR_INPUT
	bEnPgm					: BOOL;
	nValPgm					: UDINT		:= 1;
END_VAR
VAR_INPUT CONSTANT PERSISTENT
	{region 'Fixed Parameters'}
		{attribute 'parameterCategory':='Value'}
		{attribute 'TcEncoding':='UTF-8'}
		sStateText : T_BACnet_StateTextArray := BACnet_Param.sMultistate_DefaultStateText;
		
		{attribute 'parameterCategory':='EventConfig'}
		aAlarmValues : T_BACnet_MultistateValue;
		{attribute 'parameterCategory':='EventConfig'}
		aFaultValues : T_BACnet_MultistateValue;
	{endregion}
	{region 'Variable Parameters'}
		{attribute 'parameterCategory':='Value'}
		nRelinquishDefault : UDINT := 1;
		{attribute 'parameterCategory':='Value'}
		bOutOfService : BOOL;
	{endregion}
END_VAR
VAR_OUTPUT
	nPresVal			: UDINT		:= 1;
	eActPrio			: E_BACnet_Priority;			// Indicates the currently active priority of the priority array
END_VAR
VAR
	{region 'Output-Properties'}
		nStateCount			: UDINT;
	{endregion}
END_VAR

SUPER^();

METHOD PROTECTED OnObjectStateChanged
SUPER^.OnObjectStateChanged();

CASE (tState) OF
	TCOM_STATE.TCOM_STATE_PREOP:
		{warning disable C0196}
		nStateCount := F_BACnet_GetUsedStateText(sStateText);
		
		// SyncHandler:
		RequestSyncHandlers(nStateCount, nStateCount);						// Handlers for "E_BACnetPropIdentifier.PropStateText"
		_nTemp := F_BACnet_GetUsedUDINT(aAlarmValues);						// Handlers for "E_BACnetPropIdentifier.PropAlarmValues"
		RequestSyncHandlers(_nTemp, _nTemp);
		_nTemp := F_BACnet_GetUsedUDINT(aFaultValues);						// Handlers for "E_BACnetPropIdentifier.PropFaultValues"
		RequestSyncHandlers(_nTemp, _nTemp);
		RequestSyncHandlers(6, 4);											// Handlers for other properties
		{warning restore C0196}
		
		// Properties:
		EnableProperty(E_BACnetPropIdentifier.PropDeviceType, FALSE);
		
		WriteProtectProperty(E_BACnetPropIdentifier.PropNumberOfStates, TRUE);
		
		IF (BACnet_Param.bStateText_WriteProtect) THEN
			WriteProtectProperty(E_BACnetPropIdentifier.PropStateText, TRUE);
		END_IF
		
		// Ensure UTF-8 Encoding:
		F_BA_EnsureUTF8Array(ADR(sStateText), SIZEOF(T_BACnet_StateText), TO_DINT(BACnet_Param.nMultistate_StateCount));
		
	TCOM_STATE.TCOM_STATE_SAFEOP:
		SyncPropertyPvPrio(E_BACnetPropIdentifier.PropPresentValue, SIZEOF(nValPgm), ADR(nValPgm), ADR(bEnPgm), BACnet_Param.ePrio_Program, 0, eFullSync_InitPLC);
		
		SyncProperty(E_BACnetPropIdentifier.PropPresentValue, SIZEOF(nPresVal), ADR(nPresVal), 0, eSync_FromSupplement);
		SyncProperty(E_BACnetPropIdentifier.PropCurrentlyActivePriority, SIZEOF(eActPrio), ADR(eActPrio), 0, eSync_FromSupplement);
		
	TCOM_STATE.TCOM_STATE_OP:
		// Init number of used states:
		SetNumberOfStates(nStateCount);
		
		SyncProperty(E_BACnetPropIdentifier.PropRelinquishDefault, SIZEOF(nRelinquishDefault), ADR(nRelinquishDefault), 0, eFullSync_InitPLC);
		SyncProperty(E_BACnetPropIdentifier.PropOutOfService, SIZEOF(bOutOfService), ADR(bOutOfService), 0, eFullSync_InitPLC);
		SyncPropertyList(E_BACnetPropIdentifier.PropStateText, ADR(sStateText), SIZEOF(T_BACnet_StateText), nStateCount, eFullSync_InitPLC, FALSE);
		SyncPropertyList(E_BACnetPropIdentifier.PropAlarmValues, ADR(aAlarmValues), SIZEOF(UDINT), nStateCount, eFullSync_InitPLC, TRUE);
		SyncPropertyList(E_BACnetPropIdentifier.PropFaultValues, ADR(aFaultValues), SIZEOF(UDINT), nStateCount, eFullSync_InitPLC, TRUE);
		
END_CASE
END_METHOD

PROPERTY ActivePrio : E_BACnet_Priority
GET
ActivePrio := eActPrio;
END_GET
END_PROPERTY

PROPERTY StateCount : UDINT
GET
StateCount := nStateCount;
END_GET
END_PROPERTY

METHOD FB_init : BOOL
VAR_INPUT
	bInitRetains : BOOL; // if TRUE, the retain variables are initialized (warm start / cold start)
	bInCopyCode : BOOL;  // if TRUE, the instance afterwards gets moved into the copy code (online change)
END_VAR
eObjectType := E_BACnetObjType.ObjMultistateValue;
END_METHOD

END_FUNCTION_BLOCK

// POUs/Local/Objects/[Internal]/5P/FB_BACnet_MV_5P
// Multistate Value Object
// - 5 Priorities
{attribute 'pin_presentation_order_inputs' := 'bEnSfty,nValSfty,bEnCrit,nValCrit,bEnManLoc,nValManLoc,bEnPgm,nValPgm'}
{attribute 'pin_presentation_order_outputs' := 'nPresVal,eActPrio,bEvent,eRlbty'}
{attribute 'enable_dynamic_creation'}
FUNCTION_BLOCK FB_BACnet_MV_5P EXTENDS FB_BACnet_MV
VAR_INPUT
	bEnSfty					: BOOL;
	nValSfty				: UDINT		:= 1;
	bEnCrit					: BOOL;
	nValCrit				: UDINT		:= 1;
	bEnManLoc				: BOOL;
	nValManLoc				: UDINT		:= 1;
END_VAR
VAR_INPUT CONSTANT PERSISTENT
	{region 'Operational Parameters'}
		{attribute 'parameterCategory':='Manual'}
		bEnManualOperator : BOOL;
		{attribute 'parameterCategory':='Manual'}
		nValManualOperator : UDINT := 1;
	{endregion}
END_VAR

SUPER^();

METHOD PROTECTED OnObjectStateChanged
SUPER^.OnObjectStateChanged();

CASE (tState) OF
	TCOM_STATE.TCOM_STATE_PREOP:
		// SyncHandler:
		RequestSyncHandlers(4, 4);
		
	TCOM_STATE.TCOM_STATE_SAFEOP:
		SyncPropertyPvPrio(E_BACnetPropIdentifier.PropPresentValue, SIZEOF(nValSfty), ADR(nValSfty), ADR(bEnSfty), BACnet_Param.ePrio_LifeSafety, 0, eFullSync_InitPLC);
		SyncPropertyPvPrio(E_BACnetPropIdentifier.PropPresentValue, SIZEOF(nValCrit), ADR(nValCrit), ADR(bEnCrit), BACnet_Param.ePrio_Critical, 0, eFullSync_InitPLC);
		SyncPropertyPvPrio(E_BACnetPropIdentifier.PropPresentValue, SIZEOF(nValManLoc), ADR(nValManLoc), ADR(bEnManLoc), BACnet_Param.ePrio_ManLocal, 0, eFullSync_InitPLC);
		SyncPropertyPvPrio(E_BACnetPropIdentifier.PropPresentValue, SIZEOF(nValManualOperator), ADR(nValManualOperator), ADR(bEnManualOperator), BACnet_Param.ePrio_ManOperator, 0, eFullSync_InitPLC);
		
	TCOM_STATE.TCOM_STATE_OP:
		;
		
END_CASE
END_METHOD

PROPERTY EnManualOperator : BOOL
GET
EnManualOperator := bEnManualOperator;
END_GET
SET
bEnManualOperator := EnManualOperator;
END_SET
END_PROPERTY

PROPERTY ValManualOperator : UDINT
GET
ValManualOperator := nValManualOperator;
END_GET
SET
nValManualOperator := ValManualOperator;
END_SET
END_PROPERTY

END_FUNCTION_BLOCK

// POUs/Local/Objects/FB_BACnet_MV_Disp
// Multistate Setpoint Object for Setpoint
// - Used to display a value
{attribute 'enable_dynamic_creation'}
FUNCTION_BLOCK FB_BACnet_MV_Disp EXTENDS FB_BACnet_Object
VAR_INPUT
	nVal				: UDINT		:= 1;
END_VAR
VAR_INPUT CONSTANT PERSISTENT
	{region 'Fixed Parameters'}
		{attribute 'parameterCategory':='Value'}
		{attribute 'TcEncoding':='UTF-8'}
		sStateText : T_BACnet_StateTextArray := BACnet_Param.sMultistate_DefaultStateText;
	{endregion}
END_VAR
VAR_OUTPUT
	nPresVal		: UDINT		:= 1;
END_VAR
VAR
	{region 'Output-Properties'}
		nStateCount		: UDINT;
	{endregion}
END_VAR

IF bReady THEN
	nPresVal := nVal;
ELSE
	nPresVal := 1;
END_IF

SUPER^();

METHOD PROTECTED OnObjectStateChanged
SUPER^.OnObjectStateChanged();

CASE (tState) OF
	TCOM_STATE.TCOM_STATE_PREOP:
		// SyncHandler:
		{warning disable C0196}
		nStateCount := F_BACnet_GetUsedStateText(sStateText);
		{warning restore C0196}
		
		RequestSyncHandlers(nStateCount, nStateCount);						// Handlers for "E_BACnetPropIdentifier.PropStateText"
		RequestSyncHandlers(1, 1);											// Handlers for other properties
		
		// Properties:
		WriteProtectProperty(E_BACnetPropIdentifier.PropPresentValue, TRUE);
		WriteProtectProperty(E_BACnetPropIdentifier.PropNumberOfStates, TRUE);
		
		IF (BACnet_Param.bStateText_WriteProtect) THEN
			WriteProtectProperty(E_BACnetPropIdentifier.PropStateText, TRUE);
		END_IF
		
		EnableProperty(E_BACnetPropIdentifier.PropDeviceType, FALSE);
		EnableProperty(E_BACnetPropIdentifier.PropNotificationClass, FALSE);
		EnableProperty(E_BACnetPropIdentifier.PropNotifyType, FALSE);
		EnableProperty(E_BACnetPropIdentifier.PropEventEnable, FALSE);
		EnableProperty(E_BACnetPropIdentifier.PropEventTimeStamps, FALSE);
		EnableProperty(E_BACnetPropIdentifier.PropEventMessageTexts, FALSE);
		EnableProperty(E_BACnetPropIdentifier.PropEventMessageTextsConfig, FALSE);
		EnableProperty(E_BACnetPropIdentifier.PropTimeDelay, FALSE);
		EnableProperty(E_BACnetPropIdentifier.PropAckedTransitions, FALSE);
		EnableProperty(E_BACnetPropIdentifier.PropReliability, FALSE);
		EnableProperty(E_BACnetPropIdentifier.PropEventDetectionEnable, FALSE);
		EnableProperty(E_BACnetPropIdentifier.PropEventAlgorithmInhibit, FALSE);
		EnableProperty(E_BACnetPropIdentifier.PropTimeDelayNormal, FALSE);
		EnableProperty(E_BACnetPropIdentifier.PropReliabilityEvaluationInhibit, FALSE);
		EnableProperty(E_BACnetPropIdentifier.PropAlarmValues, FALSE);
		EnableProperty(E_BACnetPropIdentifier.PropFaultValues, FALSE);
		EnableProperty(E_BACnetPropIdentifier.PropRelinquishDefault, FALSE);
		EnableProperty(E_BACnetPropIdentifier.PropPriorityArray, FALSE);
		EnableProperty(E_BACnetPropIdentifier.PropCurrentlyActivePriority, FALSE);
		
		WriteProtectProperty(E_BACnetPropIdentifier.PropOutOfService, TRUE);
		// EnableProperty(E_BACnetPropIdentifier.PropStatusFlags, FALSE);
		// EnableProperty(E_BACnetPropIdentifier.PropEventState, FALSE);
		
		// Ensure UTF-8 Encoding:
		F_BA_EnsureUTF8Array(ADR(sStateText), SIZEOF(sStateText[1]), TO_DINT(BACnet_Param.nMultistate_StateCount));
		
	TCOM_STATE.TCOM_STATE_SAFEOP:
		SyncProperty(E_BACnetPropIdentifier.PropPresentValue, SIZEOF(nVal), ADR(nVal), 0, eSync_ToSupplement);
		
	TCOM_STATE.TCOM_STATE_OP:
		// Init number of used states:
		SetNumberOfStates(nStateCount);
		
		SyncPropertyList(E_BACnetPropIdentifier.PropStateText, ADR(sStateText), SIZEOF(T_BACnet_StateText), nStateCount, eFullSync_InitPLC, FALSE);

END_CASE
END_METHOD

PROPERTY StateCount : UDINT
GET
StateCount := nStateCount;
END_GET
END_PROPERTY

METHOD FB_init : BOOL
VAR_INPUT
	bInitRetains : BOOL; // if TRUE, the retain variables are initialized (warm start / cold start)
	bInCopyCode : BOOL;  // if TRUE, the instance afterwards gets moved into the copy code (online change)
END_VAR
eObjectType := E_BACnetObjType.ObjMultistateValue;
END_METHOD

END_FUNCTION_BLOCK

// POUs/Local/Objects/FB_BACnet_MV_Setp
// Multistate Setpoint Object for Setpoint
// - Used to define a setpoint by user
{attribute 'enable_dynamic_creation'}
FUNCTION_BLOCK FB_BACnet_MV_Setp EXTENDS FB_BACnet_Object
VAR_INPUT CONSTANT PERSISTENT
	{region 'Fixed Parameters'}
		{attribute 'parameterCategory':='Value'}
		{attribute 'TcEncoding':='UTF-8'}
		sStateText : T_BACnet_StateTextArray := BACnet_Param.sMultistate_DefaultStateText;
	{endregion}
	{region 'Operational Parameters'}
		{attribute 'parameterCategory':='Value'}
		nValue : UDINT := 1;
	{endregion}
END_VAR
VAR_OUTPUT
	nPresVal		: UDINT		:= 1;
END_VAR
VAR
	{region 'Output-Properties'}
		nStateCount		: UDINT;
	{endregion}
END_VAR

IF bReady THEN
	nPresVal := nValue;
ELSE
	nPresVal := 1;
END_IF

SUPER^();

METHOD PROTECTED OnObjectStateChanged
SUPER^.OnObjectStateChanged();

CASE (tState) OF
	TCOM_STATE.TCOM_STATE_PREOP:
		// SyncHandler:
		{warning disable C0196}
		nStateCount := F_BACnet_GetUsedStateText(sStateText);
		{warning restore C0196}
		
		RequestSyncHandlers(nStateCount, nStateCount);						// Handlers for "E_BACnetPropIdentifier.PropStateText"
		RequestSyncHandlers(1, 1);											// Handlers for other properties
		
		// Properties:
		WriteProtectProperty(E_BACnetPropIdentifier.PropNumberOfStates, TRUE);
		
		IF (BACnet_Param.bStateText_WriteProtect) THEN
			WriteProtectProperty(E_BACnetPropIdentifier.PropStateText, TRUE);
		END_IF
		
		EnableProperty(E_BACnetPropIdentifier.PropDeviceType, FALSE);
		EnableProperty(E_BACnetPropIdentifier.PropNotificationClass, FALSE);
		EnableProperty(E_BACnetPropIdentifier.PropNotifyType, FALSE);
		EnableProperty(E_BACnetPropIdentifier.PropEventEnable, FALSE);
		EnableProperty(E_BACnetPropIdentifier.PropEventTimeStamps, FALSE);
		EnableProperty(E_BACnetPropIdentifier.PropEventMessageTexts, FALSE);
		EnableProperty(E_BACnetPropIdentifier.PropEventMessageTextsConfig, FALSE);
		EnableProperty(E_BACnetPropIdentifier.PropTimeDelay, FALSE);
		EnableProperty(E_BACnetPropIdentifier.PropAckedTransitions, FALSE);
		EnableProperty(E_BACnetPropIdentifier.PropReliability, FALSE);
		EnableProperty(E_BACnetPropIdentifier.PropEventDetectionEnable, FALSE);
		EnableProperty(E_BACnetPropIdentifier.PropEventAlgorithmInhibit, FALSE);
		EnableProperty(E_BACnetPropIdentifier.PropTimeDelayNormal, FALSE);
		EnableProperty(E_BACnetPropIdentifier.PropReliabilityEvaluationInhibit, FALSE);
		EnableProperty(E_BACnetPropIdentifier.PropAlarmValues, FALSE);
		EnableProperty(E_BACnetPropIdentifier.PropFaultValues, FALSE);
		EnableProperty(E_BACnetPropIdentifier.PropRelinquishDefault, FALSE);
		EnableProperty(E_BACnetPropIdentifier.PropPriorityArray, FALSE);
		EnableProperty(E_BACnetPropIdentifier.PropCurrentlyActivePriority, FALSE);
		
		WriteProtectProperty(E_BACnetPropIdentifier.PropOutOfService, TRUE);
		// EnableProperty(E_BACnetPropIdentifier.PropStatusFlags, FALSE);
		// EnableProperty(E_BACnetPropIdentifier.PropEventState, FALSE);
		
		// Ensure UTF-8 Encoding:
		F_BA_EnsureUTF8Array(ADR(sStateText), SIZEOF(sStateText[1]), TO_DINT(BACnet_Param.nMultistate_StateCount));
				
	TCOM_STATE.TCOM_STATE_SAFEOP:
		;
		
	TCOM_STATE.TCOM_STATE_OP:
		// Init number of used states:
		SetNumberOfStates(nStateCount);
		
		SyncProperty(E_BACnetPropIdentifier.PropPresentValue, SIZEOF(nValue), ADR(nValue), 0, eFullSync_InitPLC);
		SyncPropertyList(E_BACnetPropIdentifier.PropStateText, ADR(sStateText), SIZEOF(T_BACnet_StateText), nStateCount, eFullSync_InitPLC, FALSE);

END_CASE
END_METHOD

PROPERTY StateCount : UDINT
GET
StateCount := nStateCount;
END_GET
END_PROPERTY

METHOD FB_init : BOOL
VAR_INPUT
	bInitRetains : BOOL; // if TRUE, the retain variables are initialized (warm start / cold start)
	bInCopyCode : BOOL;  // if TRUE, the instance afterwards gets moved into the copy code (online change)
END_VAR
eObjectType := E_BACnetObjType.ObjMultistateValue;
END_METHOD

END_FUNCTION_BLOCK

// POUs/Local/Objects/FB_BACnet_Cal
// Calendar Object
{attribute 'enable_dynamic_creation'}
FUNCTION_BLOCK FB_BACnet_Cal EXTENDS FB_BACnet_Object IMPLEMENTS I_BACnet_Cal
VAR_INPUT CONSTANT PERSISTENT
	{region 'Variable Parameters'}
		{attribute 'parameterCategory':='Value'}
		aDateList : T_BACnet_CalendarDateList;
	{endregion}
END_VAR
VAR_INPUT CONSTANT
	{region 'Variable Parameters'}
		{attribute 'parameterCategory':='Value'}
		bWriteDateList : BOOL;
	{endregion}
END_VAR
VAR_OUTPUT
	bPresVal			: BOOL;
END_VAR
VAR	
	{region 'COV'}
		bDateListChanged	: BOOL;
	{endregion}
END_VAR

IF (bWriteDateList) THEN
	WriteContent();
	bWriteDateList := FALSE;
END_IF
IF (bDateListChanged) THEN
	ReadContent();
	bDateListChanged := FALSE;
END_IF

SUPER^();

METHOD PROTECTED OnObjectStateChanged
SUPER^.OnObjectStateChanged();

CASE (tState) OF
	TCOM_STATE.TCOM_STATE_PREOP:
		// SyncHandler:
		RequestSyncHandlers(2, 0);

	TCOM_STATE.TCOM_STATE_SAFEOP:
		;
		
	TCOM_STATE.TCOM_STATE_OP:
		SyncProperty(E_BACnetPropIdentifier.PropPresentValue, SIZEOF(bPresVal), ADR(bPresVal), 0, eSync_FromSupplement);
		
		SyncPropertyCOV(E_BACnetPropIdentifier.PropDateList, ADR(bDateListChanged));
	
		WriteContent();
		
END_CASE
END_METHOD

METHOD ReadContent : BOOL
ReadContent := (ReadPropertyDateList(aDateList) = S_OK);
END_METHOD

METHOD WriteContent : BOOL
WriteContent := (WritePropertyDateList(aDateList) = S_OK);
END_METHOD

METHOD FB_init : BOOL
VAR_INPUT
	bInitRetains : BOOL; // if TRUE, the retain variables are initialized (warm start / cold start)
	bInCopyCode : BOOL;  // if TRUE, the instance afterwards gets moved into the copy code (online change)
END_VAR
eObjectType := E_BACnetObjType.ObjCalendar;
END_METHOD

END_FUNCTION_BLOCK

// POUs/Local/Objects/FB_BACnet_Device
// Device Object
{attribute 'enable_dynamic_creation'}
FUNCTION_BLOCK FB_BACnet_Device EXTENDS FB_BACnet_Object
VAR_INPUT CONSTANT PERSISTENT
	{region 'Variable Parameters'}
		{attribute 'parameterCategory':='Communication'}
		{attribute 'parameterUnit':= 'ms'}
		nAPDUSegmentTimeout : UDINT := 2000;						// (in [ms])
		{attribute 'parameterCategory':='Communication'}
		{attribute 'parameterUnit':= 'ms'}
		nAPDUTimeout : UDINT := 3000;								// (in [ms])
		{attribute 'parameterCategory':='Communication'}
		nNumberOfAPDURetries : UDINT := 3;
			 
		(*
		{attribute 'parameterCategory':='Time Synchronization'}
		bAlignIntervals : BOOL;	 
		{attribute 'parameterCategory':='Time Synchronization'}
		{attribute 'parameterUnit':= 'min'}
		nIntervalOffset : UDINT;	 
		*)		
		  
		{attribute 'parameterCategory':='General'}
		{attribute 'TcEncoding':='UTF-8'}
		sLocation : T_MaxString;
			 
		{attribute 'parameterCategory':='General'}
		{attribute 'TcEncoding':='UTF-8'}
		sApplicationSoftwareVersion : T_MaxString := 'V 1.0';	
	 
		{attribute 'parameterCategory':='General'}	
		nDatabaseRevision : UDINT;
	{endregion}
END_VAR
VAR_OUTPUT
	dtLocDateTime			: ST_BA_DateTime;
	dtLastRestoreTime 		: ST_BA_DateTime;
	dtTimeOfDeviceRestart 	: ST_BACnet_TimeStampDateTime;
	eLastRestartReason  	: E_BACnet_RestartReason;
END_VAR

SUPER^();

METHOD PROTECTED OnObjectStateChanged
SUPER^.OnObjectStateChanged();

CASE (tState) OF
	TCOM_STATE.TCOM_STATE_PREOP:
		// SyncHandler:
		RequestSyncHandlers(10, 5);
		
		// Ensure UTF-8 Encoding:
		F_BA_EnsureUTF8(ADR(sLocation), SIZEOF(sLocation));
		
	TCOM_STATE.TCOM_STATE_SAFEOP:
		;
	
	TCOM_STATE.TCOM_STATE_OP:
		SyncProperty(E_BACnetPropIdentifier.PropLocalTime, SIZEOF(dtLocDateTime.stTime), ADR(dtLocDateTime.stTime), 0, eSync_FromSupplement);
		SyncProperty(E_BACnetPropIdentifier.PropLocalDate, SIZEOF(dtLocDateTime.stDate), ADR(dtLocDateTime.stDate), 0, eSync_FromSupplement);
		SyncProperty(E_BACnetPropIdentifier.PropLastRestoreTime, SIZEOF(dtLastRestoreTime), ADR(dtLastRestoreTime), 0, eSync_FromSupplement);
		SyncProperty(E_BACnetPropIdentifier.PropTimeOfDeviceRestart, SIZEOF(dtTimeOfDeviceRestart), ADR(dtTimeOfDeviceRestart), 0, eSync_FromSupplement);
		SyncProperty(E_BACnetPropIdentifier.PropLastRestartReason, SIZEOF(eLastRestartReason), ADR(eLastRestartReason), 0, eSync_FromSupplement);

		SyncProperty(E_BACnetPropIdentifier.PropApduSegmentTimeout, SIZEOF(nAPDUSegmentTimeout), ADR(nAPDUSegmentTimeout), 0, eFullSync_InitPLC);
		SyncProperty(E_BACnetPropIdentifier.PropApduTimeout, SIZEOF(nAPDUTimeout), ADR(nAPDUTimeout), 0, eFullSync_InitPLC);
		SyncProperty(E_BACnetPropIdentifier.PropNumberOfAPDURetries, SIZEOF(nNumberOfAPDURetries), ADR(nNumberOfAPDURetries), 0, eFullSync_InitPLC);
		SyncProperty(E_BACnetPropIdentifier.PropLocation, SIZEOF(sLocation), ADR(sLocation), 0, eFullSync_InitPLC);
		SyncProperty(E_BACnetPropIdentifier.PropApplicationSoftwareVersion, SIZEOF(sApplicationSoftwareVersion), ADR(sApplicationSoftwareVersion), 0, eSync_ToSupplement);
			
		SyncProperty(E_BACnetPropIdentifier.PropDatabaseRevision, SIZEOF(nDatabaseRevision), ADR(nDatabaseRevision), 0, eSync_FromSupplement);
		
END_CASE
END_METHOD

PROPERTY Location : T_MaxString
GET
Location:=sLocation;
END_GET
SET
sLocation:=Location;
END_SET
END_PROPERTY

METHOD FB_init : BOOL
VAR_INPUT
	bInitRetains : BOOL; // if TRUE, the retain variables are initialized (warm start / cold start)
	bInCopyCode : BOOL;  // if TRUE, the instance afterwards gets moved into the copy code (online change)
END_VAR
eObjectType := E_BACnetObjType.ObjDevice;
END_METHOD

END_FUNCTION_BLOCK

// POUs/Local/Objects/FB_BACnet_Loop
// Loop Object
{attribute 'enable_dynamic_creation'}
FUNCTION_BLOCK FB_BACnet_Loop EXTENDS FB_BACnet_BaseLoop
VAR_INPUT
	fSetpoint				: REAL;
	fCtrlVar				: REAL;
END_VAR

SUPER^();

METHOD PROTECTED OnObjectStateChanged
SUPER^.OnObjectStateChanged();

CASE (tState) OF
	TCOM_STATE.TCOM_STATE_PREOP:
		// SyncHandler:
		RequestSyncHandlers(0, 2);
		
		// Properties:
		WriteProtectProperty(E_BACnetPropIdentifier.PropManipulatedVariableReference, TRUE);
		WriteProtectProperty(E_BACnetPropIdentifier.PropControlledVariableReference, TRUE);
		WriteProtectProperty(E_BACnetPropIdentifier.PropSetpointReference, TRUE);
		WriteProtectProperty(E_BACnetPropIdentifier.PropPriorityForWriting, TRUE);
		
	TCOM_STATE.TCOM_STATE_SAFEOP:
		SyncProperty(E_BACnetPropIdentifier.PropSetpoint, SIZEOF(fSetpoint), ADR(fSetpoint), 0, eSync_ToSupplement);
		SyncProperty(E_BACnetPropIdentifier.PropControlledVariableValue, SIZEOF(fCtrlVar), ADR(fCtrlVar), 0, eSync_ToSupplement);
	
END_CASE
END_METHOD

PROPERTY ControlledVariable : REAL
GET
ControlledVariable := fCtrlVar;
END_GET
END_PROPERTY

PROPERTY Setpoint : REAL
GET
Setpoint := fSetpoint;
END_GET
END_PROPERTY

END_FUNCTION_BLOCK

// POUs/Local/Objects/[Base]/FB_BACnet_BaseLoop
// Loop Object
{attribute 'enable_dynamic_creation'}
FUNCTION_BLOCK ABSTRACT FB_BACnet_BaseLoop EXTENDS FB_BACnet_EventObject
VAR_INPUT
	bEn						: BOOL;
	
	bEnSync					: BOOL;
	fValSync				: REAL;
END_VAR
VAR_INPUT CONSTANT PERSISTENT
	{region 'Variable Parameters'}
		{attribute 'parameterCategory':='Value'}
		bOutOfService : BOOL;
		{attribute 'parameterCategory':='Value'}
		fCOVIncrement : REAL := 0.1;
		{attribute 'parameterCategory':='Value'}
		eOutputUnit : E_BA_Unit := E_BA_Unit.eOther_Percent;
		
		{attribute 'parameterCategory':='Config'}
		eOpMode : E_BA_PIDMode := E_BA_PIDMode.eP1ID;
		{attribute 'parameterCategory':='Config'}
		eAction : E_BA_Action := E_BA_Action.eDirect;
		{attribute 'parameterCategory':='Config'}
		fBias : REAL := 0;
		{attribute 'parameterCategory':='Config'}
		fMinOutput : REAL := 0;
		{attribute 'parameterCategory':='Config'}
		fMaxOutput : REAL := 100;
		{attribute 'parameterCategory':='Config'}
		{attribute 'parameterUnit':= '1/s'}
		fAccLimit : REAL := 0.0;							// Setpoint acceleration limit positive and negative [1/s]
		{attribute 'parameterCategory':='Config'}
		fProportionalConstant : REAL := 1;
		{attribute 'parameterCategory':='Config'}
		eProportionalConstantUnit : E_BA_Unit := E_BA_Unit.eOther_NoUnits;
		{attribute 'parameterCategory':='Config'}
		fIntegralConstant : REAL := 60;
		{attribute 'parameterCategory':='Config'}
		eIntegralConstantUnit : E_BA_Unit := E_BA_Unit.eTime_Seconds;
		{attribute 'parameterCategory':='Config'}
		fDerivativeConstant : REAL := 0;
		{attribute 'parameterCategory':='Config'}
		eDerivativeConstantUnit : E_BA_Unit := E_BA_Unit.eTime_Seconds;
		
		{attribute 'parameterCategory':='EventConfig'}
		fDeadband : REAL := 0.1;
		{attribute 'parameterCategory':='EventConfig'}
		fErrorLimit : REAL := 0;
	{endregion}
END_VAR
VAR_OUTPUT
	fPresVal				: REAL;
END_VAR
VAR
	{region 'Output-Properties'}
		fPropBand			: REAL; 						// Controller output in range of -100...100% in relation to Min.-/Max.-output
	{endregion}
END_VAR
VAR
	{region 'Internal'}
		{attribute 'conditionalshow'}
		fbPIDCtrl			: FB_BA_PIDCtrl;
		{attribute 'conditionalshow'}
		fbAccLimit			: FB_BACnet_AccLimit;
		{attribute 'hide'}
		rfOoS				: FB_BA_RFTrig;
	{endregion}
END_VAR

IF (bReady) THEN
	rfOoS(bValue:=stStatusFlags.bOutOfService);
	IF (NOT rfOoS.bValue) THEN
		// Update functional settings:
		fbPIDCtrl.bEn := (bEn) AND_THEN (eRlbty = E_BA_Reliability.eNoFaultDetected);
		fbPIDCtrl.fW := Setpoint;
		fbPIDCtrl.fX := ControlledVariable;
		fbPIDCtrl.eActn := eAction;
			
		// Update configuration settings:
		IF (fbPIDCtrl.bEn) THEN
			fbPIDCtrl.fYMin := fMinOutput;
			fbPIDCtrl.fYMax := fMaxOutput;
			fbPIDCtrl.fProportionalConstant := fProportionalConstant;
			fbPIDCtrl.tIntegralTime := (TO_TIME(fIntegralConstant) * BAComn_Global.nMilli2Sek);
			fbPIDCtrl.tDerivativeTime := (TO_TIME(fDerivativeConstant) * BAComn_Global.nMilli2Sek);
			fbPIDCtrl.eOperationMode := eOpMode;
			fbPIDCtrl.fNeutralZone := fDeadband;
			
			IF (bEnSync) THEN
				fbPIDCtrl.bSync := TRUE;
				fbPIDCtrl.fSync := fValSync;
			ELSIF (rfOoS.Qf) THEN
				fbPIDCtrl.bSync := TRUE;
				fbPIDCtrl.fSync := fPresVal;	// Synchronize with last (may manipulated by operator) present value
			ELSE
				fbPIDCtrl.bSync := FALSE;
				fbPIDCtrl.fSync := 0;
			END_IF
		END_IF
		
		fbPIDCtrl();
	
		// Limit present value:
		fbAccLimit(X:=fbPIDCtrl.fY, Amax:=fAccLimit, Y=>fPresVal);
		
		// Calculate proportional band:
		IF (fMaxOutput > 0.0) AND (fMinOutput >= 0.0) THEN
			fPropBand := ((fPresVal - fMinOutput) / (fMaxOutput - fMinOutput)) * 100.0;
		ELSIF (fMaxOutput <= 0.0) AND (fMinOutput < 0.0) THEN
			fPropBand := ((fPresVal - fMaxOutput) / (fMaxOutput - fMinOutput)) * 100.0;
		ELSIF (fPresVal > 0.0) AND (fMaxOutput > 0.0) THEN
			fPropBand := (fPresVal / fMaxOutput) * 100.0;
		ELSIF (fPresVal < 0.0) AND (fMinOutput < 0.0) THEN
			fPropBand := (fPresVal / fMinOutput) * -100.0;
		ELSE
			fPropBand := 0.0;
		END_IF
	END_IF
END_IF

SUPER^();

METHOD PROTECTED OnObjectStateChanged
SUPER^.OnObjectStateChanged();

CASE (tState) OF
	TCOM_STATE.TCOM_STATE_PREOP:
		// SyncHandler:
		RequestSyncHandlers(16, 16);
		
		// Properties:
		WriteProtectProperty(E_BACnetPropIdentifier.PropPresentValue, TRUE);
		WriteProtectProperty(E_BACnetPropIdentifier.PropSetpoint, TRUE);
		WriteProtectProperty(E_BACnetPropIdentifier.PropControlledVariableValue, TRUE);
		
	TCOM_STATE.TCOM_STATE_SAFEOP:
		SyncProperty(E_BACnetPropIdentifier.PropPresentValue, SIZEOF(fPresVal), ADR(fPresVal), 0, eFullSync_InitPLC);
	
	TCOM_STATE.TCOM_STATE_OP:
		SyncProperty(E_BACnetPropIdentifier.PropOutputUnits, SIZEOF(eOutputUnit), ADR(eOutputUnit), 0, eFullSync_InitPLC);
		SyncProperty(E_BACnetPropIdentifier.PropOutOfService, SIZEOF(bOutOfService), ADR(bOutOfService), 0, eFullSync_InitPLC);
		SyncProperty(E_BACnetPropIdentifier.PropCovIncrement, SIZEOF(fCOVIncrement), ADR(fCOVIncrement), 0, eFullSync_InitPLC);
		SyncProperty(E_BACnetPropIdentifier.PropProportionalConstant, SIZEOF(fProportionalConstant), ADR(fProportionalConstant), 0, eFullSync_InitPLC);
		SyncProperty(E_BACnetPropIdentifier.PropProportionalConstantUnits, SIZEOF(eProportionalConstantUnit), ADR(eProportionalConstantUnit), 0, eFullSync_InitPLC);
		SyncProperty(E_BACnetPropIdentifier.PropIntegralConstant, SIZEOF(fIntegralConstant), ADR(fIntegralConstant), 0, eFullSync_InitPLC);
		SyncProperty(E_BACnetPropIdentifier.PropIntegralConstantUnits, SIZEOF(eIntegralConstantUnit), ADR(eIntegralConstantUnit), 0, eFullSync_InitPLC);
		SyncProperty(E_BACnetPropIdentifier.PropDerivativeConstant, SIZEOF(fDerivativeConstant), ADR(fDerivativeConstant), 0, eFullSync_InitPLC);
		SyncProperty(E_BACnetPropIdentifier.PropDerivativeConstantUnits, SIZEOF(eDerivativeConstantUnit), ADR(eDerivativeConstantUnit), 0, eFullSync_InitPLC);
		SyncProperty(E_BACnetPropIdentifier.PropDeadband, SIZEOF(fDeadband), ADR(fDeadband), 0, eFullSync_InitPLC);
		SyncProperty(E_BACnetPropIdentifier.PropErrorLimit, SIZEOF(fErrorLimit), ADR(fErrorLimit), 0, eFullSync_InitPLC);
		SyncProperty(E_BACnetPropIdentifier.PropMinimumOutput, SIZEOF(fMinOutput), ADR(fMinOutput), 0, eFullSync_InitPLC);
		SyncProperty(E_BACnetPropIdentifier.PropMaximumOutput, SIZEOF(fMaxOutput), ADR(fMaxOutput), 0, eFullSync_InitPLC);
		SyncProperty(E_BACnetPropIdentifier.PropActionProp, SIZEOF(eAction), ADR(eAction), 0, eFullSync_InitPLC);
		SyncProperty(E_BACnetPropIdentifier.PropBias, SIZEOF(fBias), ADR(fBias), 0, eFullSync_InitPLC);
		
		WritePropertyUDInt(E_BACnetPropIdentifier.PropPriorityForWriting, BACnet_Param.nLoop_PrioForWriting);
		
END_CASE
END_METHOD

PROPERTY ABSTRACT ControlledVariable : REAL
GET
END_GET
END_PROPERTY

PROPERTY ProportionalBand : REAL
GET
ProportionalBand := fPropBand;
END_GET
END_PROPERTY

PROPERTY ABSTRACT Setpoint : REAL
GET
END_GET
END_PROPERTY

METHOD FB_init : BOOL
VAR_INPUT
	bInitRetains : BOOL; // if TRUE, the retain variables are initialized (warm start / cold start)
	bInCopyCode : BOOL;  // if TRUE, the instance afterwards gets moved into the copy code (online change)
END_VAR
eObjectType := E_BACnetObjType.ObjLoop;
END_METHOD

END_FUNCTION_BLOCK

// POUs/Helper/FB_BACnet_AccLimit
FUNCTION_BLOCK FB_BACnet_AccLimit
VAR_INPUT
	X : REAL; (* input value [1] *)
	Amax : REAL; (* maximum acceleration of X [1/s]; 0 = limit disabled *)
	TiCycle : REAL; (* cycle time [s] of task; 0 = use internal measuring *)
END_VAR
VAR_OUTPUT
	Y : REAL; (* limited X value [1] *)
	A : REAL; (* input acceleration [1/s] *)
END_VAR
VAR
	_sysTime	: GETCPUCOUNTER;
	_Time		: T_LARGE_INTEGER;
	_TimeOld	: T_LARGE_INTEGER;
	_tCycleTime	: REAL;
	_bFirstScan	: BOOL:=TRUE;
	_foldY		: REAL;
END_VAR

(* determine cycle time *)
IF TiCycle = 0.0 THEN
	_TimeOld := _Time;
	_sysTime(cpuCntLoDW=> _Time.dwLowPart, cpuCntHiDW=> _Time.dwHighPart);
	_tCycleTime := F_BACnet_SysTimeDiff(In1:=_Time, In2:=_TimeOld);
ELSE
	_tCycleTime := TiCycle;
END_IF

IF (NOT _bFirstScan) THEN
	(* exit on wrong cycle time *)
	IF _tCycleTime <= 0.0 THEN
		RETURN;
	END_IF
	(* calculate current acceleration *)
	A := (X - _foldY) / _tCycleTime;
	IF (Amax <> 0.0) THEN
		Amax := ABS(Amax);
		IF (ABS(A) > Amax) THEN
			IF (A >= 0.0) THEN
				Y := _foldY + (Amax * _tCycleTime);
			ELSE
				Y := _foldY - (Amax * _tCycleTime);
			END_IF
		ELSE
			Y := X;
		END_IF
	ELSE
		Y := X;
	END_IF
ELSE
	Y := X;
END_IF

_foldY := Y;
_bFirstScan:=FALSE;

END_FUNCTION_BLOCK

// POUs/Helper/[internal]/F_BACnet_SysTimeDiff
{attribute 'hide'}
FUNCTION F_BACnet_SysTimeDiff : REAL
VAR_INPUT
	In1, In2 : T_LARGE_INTEGER;
END_VAR

F_BACnet_SysTimeDiff := LREAL_TO_REAL(INT64_TO_LREAL(Int64Sub64(In1, In2)) / 10000000.0); (* [s] *)

END_FUNCTION

// POUs/Local/Objects/FB_BACnet_NC
// Notification Class Object
{attribute 'enable_dynamic_creation'}
FUNCTION_BLOCK FB_BACnet_NC EXTENDS FB_BACnet_Object
VAR_INPUT CONSTANT PERSISTENT
	{region 'Variable Parameters'}
		{attribute 'parameterCategory':='Config'}
		nNotificationClass : UDINT;
		{attribute 'parameterCategory':='Config'}
		aPriority : T_BACnet_EventTransitionPriority;
		{attribute 'parameterCategory':='Config'}
		aAckRequired : T_BACnet_EventTransitions;
		{attribute 'parameterCategory':='Config'}
		aRecipientList : T_BACnet_RecipientList;
	{endregion}
END_VAR
VAR_INPUT CONSTANT
	{region 'Variable Parameters'}
		{attribute 'parameterCategory':='Config'}
		bWriteRecipientList : BOOL;
	{endregion}
END_VAR
VAR
	{region 'COV'}
		bRecipientListChanged : BOOL;
	{endregion}
END_VAR

SUPER^();

IF (bWriteRecipientList) THEN
	bWriteRecipientList := FALSE;
	WritePropertyRecipientList(aRecipientList);
END_IF
IF (bRecipientListChanged) THEN
	bRecipientListChanged := FALSE;
	ReadPropertyRecipientList(aRecipientList);
END_IF

METHOD PROTECTED OnObjectStateChanged
SUPER^.OnObjectStateChanged();

CASE (tState) OF
	TCOM_STATE.TCOM_STATE_PREOP:
		// SyncHandler:
		RequestSyncHandlers(8, 7);
		
	TCOM_STATE.TCOM_STATE_SAFEOP:
		;
		
	TCOM_STATE.TCOM_STATE_OP:
		IF (SyncPropertyCOV(E_BACnetPropIdentifier.PropRecipientList, ADR(bRecipientListChanged))) THEN
			WritePropertyRecipientList(aRecipientList);
		END_IF
		
		SyncProperty(E_BACnetPropIdentifier.PropNotificationClass, SIZEOF(nNotificationClass), ADR(nNotificationClass), 0, eFullSync_InitPLC);
		SyncPropertyIdx(E_BACnetPropIdentifier.PropPriority, SIZEOF(UDINT), ADR(aPriority[E_BA_EventTransition.eToOffnormal]), (E_BACnet_EventTransitionBits.eToOffnormal+1), 0, eFullSync_InitPLC);	
		SyncPropertyIdx(E_BACnetPropIdentifier.PropPriority, SIZEOF(UDINT), ADR(aPriority[E_BA_EventTransition.eToFault]), (E_BACnet_EventTransitionBits.eToFault+1), 0, eFullSync_InitPLC);	
		SyncPropertyIdx(E_BACnetPropIdentifier.PropPriority, SIZEOF(UDINT), ADR(aPriority[E_BA_EventTransition.eToNormal]), (E_BACnet_EventTransitionBits.eToNormal+1), 0, eFullSync_InitPLC);
		SyncPropertyIdx(E_BACnetPropIdentifier.PropAckRequired, SIZEOF(BOOL), ADR(aAckRequired[E_BA_EventTransition.eToOffnormal]), E_BACnet_EventTransitionBits.eToOffnormal, 0, eFullSync_InitPLC);	
		SyncPropertyIdx(E_BACnetPropIdentifier.PropAckRequired, SIZEOF(BOOL), ADR(aAckRequired[E_BA_EventTransition.eToFault]), E_BACnet_EventTransitionBits.eToFault, 0, eFullSync_InitPLC);	
		SyncPropertyIdx(E_BACnetPropIdentifier.PropAckRequired, SIZEOF(BOOL), ADR(aAckRequired[E_BA_EventTransition.eToNormal]), E_BACnet_EventTransitionBits.eToNormal, 0, eFullSync_InitPLC);
		
END_CASE
END_METHOD

METHOD FB_init : BOOL
VAR_INPUT
	bInitRetains : BOOL; // if TRUE, the retain variables are initialized (warm start / cold start)
	bInCopyCode : BOOL;  // if TRUE, the instance afterwards gets moved into the copy code (online change)
END_VAR
eObjectType := E_BACnetObjType.ObjNotificationClass;
END_METHOD

END_FUNCTION_BLOCK

// POUs/Local/Objects/FB_BACnet_Prog
// Program Object
{attribute 'enable_dynamic_creation'}
FUNCTION_BLOCK FB_BACnet_Prog EXTENDS FB_BACnet_Object
VAR_OUTPUT
	eState			: E_BACnet_ProgramState;
END_VAR

SUPER^();

METHOD PROTECTED OnObjectStateChanged
SUPER^.OnObjectStateChanged();

CASE (tState) OF
	TCOM_STATE.TCOM_STATE_PREOP:
		// SyncHandler:
		RequestSyncHandlers(1, 0);
		
	TCOM_STATE.TCOM_STATE_SAFEOP:
		;
	
	TCOM_STATE.TCOM_STATE_OP:
		SyncProperty(E_BACnetPropIdentifier.PropProgramState, SIZEOF(eState), ADR(eState), 0, eSync_FromSupplement);
		
END_CASE
END_METHOD

METHOD FB_init : BOOL
VAR_INPUT
	bInitRetains : BOOL; // if TRUE, the retain variables are initialized (warm start / cold start)
	bInCopyCode : BOOL;  // if TRUE, the instance afterwards gets moved into the copy code (online change)
END_VAR
eObjectType := E_BACnetObjType.ObjProg;
END_METHOD

END_FUNCTION_BLOCK

// POUs/Local/Objects/FB_BACnet_SchedA
// Analog Scheduler Object
{attribute 'enable_dynamic_creation'}
FUNCTION_BLOCK FB_BACnet_SchedA EXTENDS FB_BACnet_BaseSched
VAR_INPUT CONSTANT PERSISTENT
	{region 'Fixed Parameters'}
		{attribute 'parameterCategory':='Value'}
		fScheduleDefault : REAL;
	{endregion}
END_VAR
VAR_OUTPUT
	fPresVal		: REAL;
END_VAR

SUPER^();

METHOD PROTECTED OnObjectStateChanged
SUPER^.OnObjectStateChanged();

CASE (tState) OF
	TCOM_STATE.TCOM_STATE_PREOP:
		// SyncHandler:
		RequestSyncHandlers(1, 6);
		
	TCOM_STATE.TCOM_STATE_SAFEOP:
		;	
		
	TCOM_STATE.TCOM_STATE_OP:
		SyncProperty(E_BACnetPropIdentifier.PropPresentValueReal, SIZEOF(fPresVal), ADR(fPresVal), 0, eSync_FromSupplement);	
		WritePropertyValueEx(E_BACnetPropIdentifier.PropScheduleDefault, eDatatype, SIZEOF(fScheduleDefault), ADR(fScheduleDefault));
		
END_CASE
END_METHOD

METHOD FB_init : BOOL
VAR_INPUT
	bInitRetains : BOOL; // if TRUE, the retain variables are initialized (warm start / cold start)
	bInCopyCode : BOOL;  // if TRUE, the instance afterwards gets moved into the copy code (online change)
END_VAR
eDatatype := E_BACnet_ValueChoice.eRealValue;

// Init default values:
aWeek := F_BACnet_SchedWeekly1xA(E_BA_Weekday.eMonday, E_BA_Weekday.eFriday, T#0H, 0.0);
END_METHOD

END_FUNCTION_BLOCK

// POUs/Local/Objects/[Base]/FB_BACnet_BaseSched
FUNCTION_BLOCK ABSTRACT FB_BACnet_BaseSched EXTENDS FB_BACnet_Object
VAR_INPUT CONSTANT PERSISTENT
	{region 'Variable Parameters'}
		{attribute 'parameterCategory':='Value'}
		aWeek : T_BACnet_SchedWeek;															// Entries (separated per days) for weekly organization
		{attribute 'parameterCategory':='Value'}
		aCalendar : T_BACnet_SchedCalendar;													// Entries (separated per calendar) for global (calendar) exceptions organization (See "fbCalendar")
		{attribute 'parameterCategory':='Value'}
		aException : T_BACnet_SchedExceptionList;											// Entries (separated per exception count) for local (Presrent instance) exceptions organization
		{attribute 'parameterCategory':='Value'}
		bOutOfService : BOOL;
			 
		{attribute 'parameterCategory':='Config'}
		aObjectPropertyReferences : ARRAY[1 .. BACnet_Param.nSched_ReferenceCount] OF ST_BACnet_ObjectPropertyReference;
	{endregion}
END_VAR
VAR_INPUT CONSTANT
	{region 'Variable Parameters'}
		{attribute 'parameterCategory':='Value'}
		bWriteWeekly : BOOL;
		{attribute 'parameterCategory':='Value'}
		bWriteException : BOOL;
	{endregion}
END_VAR
VAR_OUTPUT
	eRlbty				: E_BA_Reliability;
END_VAR
VAR	
	{region 'Event'}
		stStatusFlags			: ST_BA_StatusFlags;
	{endregion}
	{region 'COV'}
		bWeeklyChanged			: BOOL;
		bExceptionChanged		: BOOL;
	{endregion}
END_VAR
VAR
	{region 'Internal'}
		eDatatype				: E_BACnet_ValueChoice					:= E_BACnet_ValueChoice.eNullValue;
	{endregion}
END_VAR

IF (bWriteWeekly OR bWriteException) THEN
	WriteContent(bWriteWeekly, bWriteException);
	
	bWriteWeekly := FALSE;
	bWriteException := FALSE;
END_IF
IF (bWeeklyChanged OR bExceptionChanged) THEN
	ReadContent(bWeeklyChanged, bExceptionChanged);
	
	bWeeklyChanged := FALSE;
	bExceptionChanged := FALSE;
END_IF

SUPER^();

METHOD PROTECTED OnObjectStateChanged
VAR
	i : DINT;
	_bResult : BOOL;
END_VAR
SUPER^.OnObjectStateChanged();

CASE (tState) OF
	TCOM_STATE.TCOM_STATE_PREOP:
		// SyncHandler:
		RequestSyncHandlers(8, 1);
		
		// Properties:
		WriteProtectProperty(E_BACnetPropIdentifier.PropScheduleDefault, TRUE);
	
	TCOM_STATE.TCOM_STATE_SAFEOP:
		;
		
	TCOM_STATE.TCOM_STATE_OP:
		// Validate referred properties:
		FOR i:= 1 TO TO_DINT(BACnet_Param.nSched_ReferenceCount) DO
			ValidateReference(aObjectPropertyReferences[i].iObject, aObjectPropertyReferences[i].tObjectID, 16#FF);
		END_FOR
		ObjectPropertyReferences := aObjectPropertyReferences;
		
		SyncPropertyCOV(E_BACnetPropIdentifier.PropWeeklySchedule, ADR(bWeeklyChanged));
		SyncPropertyCOV(E_BACnetPropIdentifier.PropExceptionSchedule, ADR(bExceptionChanged));
	
		SyncProperty(E_BACnetPropIdentifier.PropOutOfService, SIZEOF(bOutOfService), ADR(bOutOfService), 0, eFullSync_InitPLC);
		
		SyncPropertyIdx(E_BACnetPropIdentifier.PropStatusFlags, SIZEOF(BOOL), ADR(stStatusFlags.bOverridden), E_BACnet_StatusFlags.eOverridden, 0, eSync_FromSupplement);	
		SyncPropertyIdx(E_BACnetPropIdentifier.PropStatusFlags, SIZEOF(BOOL), ADR(stStatusFlags.bOutOfService), E_BACnet_StatusFlags.eOutOfService, 0, eSync_FromSupplement);	
		SyncPropertyIdx(E_BACnetPropIdentifier.PropStatusFlags, SIZEOF(BOOL), ADR(stStatusFlags.bFault), E_BACnet_StatusFlags.eFault, 0, eSync_FromSupplement);	
		SyncPropertyIdx(E_BACnetPropIdentifier.PropStatusFlags, SIZEOF(BOOL), ADR(stStatusFlags.bInAlarm), E_BACnet_StatusFlags.eInAlarm, 0, eSync_FromSupplement);
		SyncProperty(E_BACnetPropIdentifier.PropReliability, SIZEOF(eRlbty), ADR(eRlbty), 0, eSync_FromSupplement);

		WriteContent(TRUE, TRUE);
		WritePropertyUDInt(E_BACnetPropIdentifier.PropPriorityForWriting, BACnet_Param.nSched_PrioForWriting);
		
END_CASE
END_METHOD

METHOD ReadContent : BOOL
VAR_INPUT
	bWeeklySched		: BOOL		:= TRUE;
	bExceptSched		: BOOL		:= TRUE;
END_VAR
IF (bWeeklySched) THEN
	IF (ReadPropertyWeeklySched(aWeek, eDataType) <> S_OK) THEN
		RETURN;
	END_IF
END_IF
IF (bExceptSched) THEN
	IF (ReadPropertyExceptionSched(aCalendar, aException, eDataType) <> S_OK) THEN
		RETURN;
	END_IF
END_IF

ReadContent := TRUE;
END_METHOD

METHOD WriteContent : BOOL
VAR_INPUT
	bWeeklySched		: BOOL		:= TRUE;
	bExceptSched		: BOOL		:= TRUE;
END_VAR
WriteContent := TRUE;

IF (bWeeklySched) THEN
	_hResult := WritePropertyWeeklySched(aWeek, eDataType);
	WriteContent := (WriteContent) AND (_hResult=S_OK);
	bWeeklyChanged := FALSE;
END_IF
IF (bExceptSched) THEN
	_hResult := WritePropertyExceptionSched(aCalendar, aException, eDataType);
	WriteContent := (WriteContent) AND (_hResult=S_OK);
	bExceptionChanged := FALSE;
END_IF
END_METHOD

PROPERTY ObjectPropertyReferences : ARRAY[1 .. BACnet_Param.nSched_ReferenceCount] OF ST_BACnet_ObjectPropertyReference
GET
ObjectPropertyReferences := aObjectPropertyReferences;
END_GET
SET
aObjectPropertyReferences := ObjectPropertyReferences;

{warning disable C0196}
WritePropertyReferenceList(E_BACnetPropIdentifier.PropListOfObjectPropertyReferences, aObjectPropertyReferences);
{warning restore C0196}
END_SET
END_PROPERTY

METHOD FB_init : BOOL
VAR_INPUT
	bInitRetains : BOOL; // if TRUE, the retain variables are initialized (warm start / cold start)
	bInCopyCode : BOOL;  // if TRUE, the instance afterwards gets moved into the copy code (online change)
END_VAR
eObjectType := E_BACnetObjType.ObjSchedule;
END_METHOD

END_FUNCTION_BLOCK

// POUs/Helper/Schedule/Weekly/F_BACnet_SchedWeekly1xA
// Returns an initialized analog weekly scheduler.
FUNCTION F_BACnet_SchedWeekly1xA : T_BACnet_SchedWeek
VAR_INPUT
	eDayFrom	: E_BA_Weekday		:= E_BA_Weekday.eMonday;
	eDayTo		: E_BA_Weekday		:= E_BA_Weekday.eSunday;
	
	tTime1		: TIME;
	fValue1		: REAL;
END_VAR

F_BA_SetWeekdays(F_BACnet_SchedWeekly1xA, eDayFrom, eDayTo, 1, tTime1, F_BA_RVal(fValue1));

END_FUNCTION

// POUs/Local/Objects/FB_BACnet_SchedB
// Binary Scheduler Object
{attribute 'enable_dynamic_creation'}
FUNCTION_BLOCK FB_BACnet_SchedB EXTENDS FB_BACnet_BaseSched
VAR_INPUT
	{attribute 'parameterUnit':= 's'}
	nPredTime : UDINT;
END_VAR
VAR_INPUT CONSTANT PERSISTENT
	{region 'Fixed Parameters'}
		{attribute 'parameterCategory':='Value'}
		bScheduleDefault 	: BOOL;
	{endregion}
END_VAR
VAR_OUTPUT
	bPresVal				: BOOL;
	bPredVal				: BOOL;
END_VAR

SUPER^();

METHOD PROTECTED OnObjectStateChanged
VAR
	_ePropPresentVal		: E_BACnetPropIdentifier;
END_VAR
SUPER^.OnObjectStateChanged();

CASE (tState) OF
	TCOM_STATE.TCOM_STATE_PREOP:
		// SyncHandler:
		RequestSyncHandlers(2, 1);
		
	TCOM_STATE.TCOM_STATE_SAFEOP:
		;
		
	TCOM_STATE.TCOM_STATE_OP:
		CASE (eDatatype) OF
			E_BACnet_ValueChoice.eEnumerationValue:
				_ePropPresentVal := E_BACnetPropIdentifier.PropPresentValueEnumerated;
			E_BACnet_ValueChoice.eBoolValue:
				_ePropPresentVal := E_BACnetPropIdentifier.PropPresentValueBool;
		ELSE
			iOwner.LogMsg.Show1(ADSLOG_MSGTYPE_ERROR, 'OOSC17', 'Property-synchronization aborted: Invalid datatype "%d"!', F_INT(eDatatype), FALSE);		
			RETURN;
		END_CASE

		SyncProperty(_ePropPresentVal, SIZEOF(bPresVal), ADR(bPresVal), 0, eSync_FromSupplement);
		SyncProperty(E_BACnetPropIdentifier.PropPredictedScheduleBoolValue, SIZEOF(bPredVal), ADR(bPredVal), 0, eSync_FromSupplement);

		SyncProperty(E_BACnetPropIdentifier.PropPredictScheduleValueTime, SIZEOF(nPredTime), ADR(nPredTime), 0, eSync_ToSupplement);

		WritePropertyValueEx(E_BACnetPropIdentifier.PropScheduleDefault, eDatatype, SIZEOF(bScheduleDefault), ADR(bScheduleDefault));
		
END_CASE
END_METHOD

METHOD FB_init : BOOL
VAR_INPUT
	bInitRetains : BOOL; // if TRUE, the retain variables are initialized (warm start / cold start)
	bInCopyCode : BOOL;  // if TRUE, the instance afterwards gets moved into the copy code (online change)
END_VAR
CASE (BACnet_Param.eSched_BType) OF
	E_BACnet_SchedBType.eBinaryPV:
		eDatatype := E_BACnet_ValueChoice.eEnumerationValue;
	E_BACnet_SchedBType.eBool:
		eDatatype := E_BACnet_ValueChoice.eBoolValue;
END_CASE

// Init default values:
aWeek := F_BACnet_SchedWeekly1xB(E_BA_Weekday.eMonday, E_BA_Weekday.eFriday, T#0H, FALSE);
END_METHOD

END_FUNCTION_BLOCK

// POUs/Helper/Schedule/Weekly/F_BACnet_SchedWeekly1xB
// Returns an initialized binary weekly scheduler.
FUNCTION F_BACnet_SchedWeekly1xB : T_BACnet_SchedWeek
VAR_INPUT
	eDayFrom	: E_BA_Weekday		:= E_BA_Weekday.eMonday;
	eDayTo		: E_BA_Weekday		:= E_BA_Weekday.eSunday;
	
	tTime1		: TIME;
	bValue1		: BOOL;
END_VAR

F_BA_SetWeekdays(F_BACnet_SchedWeekly1xB, eDayFrom, eDayTo, 1, tTime1, F_BA_BVal(bValue1));

END_FUNCTION

// POUs/Local/Objects/FB_BACnet_SchedM
// Multistate Scheduler Object
{attribute 'enable_dynamic_creation'}
FUNCTION_BLOCK FB_BACnet_SchedM EXTENDS FB_BACnet_BaseSched
VAR_INPUT CONSTANT PERSISTENT
	{region 'Fixed Parameters'}
		{attribute 'parameterCategory':='Value'}
		nScheduleDefault : UDINT;
	{endregion}
END_VAR
VAR_OUTPUT
	nPresVal		: UDINT;
END_VAR

SUPER^();

METHOD PROTECTED OnObjectStateChanged
SUPER^.OnObjectStateChanged();

CASE (tState) OF
	TCOM_STATE.TCOM_STATE_PREOP:
		// SyncHandler:
		RequestSyncHandlers(1, 0);
		
	TCOM_STATE.TCOM_STATE_SAFEOP:
		;
		
	TCOM_STATE.TCOM_STATE_OP:
		SyncProperty(E_BACnetPropIdentifier.PropPresentValueUnsigned, SIZEOF(nPresVal), ADR(nPresVal), 0, eSync_FromSupplement);
		
		WritePropertyValueEx(E_BACnetPropIdentifier.PropScheduleDefault, eDatatype, SIZEOF(nScheduleDefault), ADR(nScheduleDefault));
		
END_CASE
END_METHOD

METHOD FB_init : BOOL
VAR_INPUT
	bInitRetains : BOOL; // if TRUE, the retain variables are initialized (warm start / cold start)
	bInCopyCode : BOOL;  // if TRUE, the instance afterwards gets moved into the copy code (online change)
END_VAR
eDatatype := E_BACnet_ValueChoice.eUnsignedValue;

// Init default values:
aWeek := F_BACnet_SchedWeekly1xM(E_BA_Weekday.eMonday, E_BA_Weekday.eFriday, T#0H, 1);
END_METHOD

END_FUNCTION_BLOCK

// POUs/Helper/Schedule/Weekly/F_BACnet_SchedWeekly1xM
// Returns an initialized multistate weekly scheduler.
FUNCTION F_BACnet_SchedWeekly1xM : T_BACnet_SchedWeek
VAR_INPUT
	eDayFrom	: E_BA_Weekday		:= E_BA_Weekday.eMonday;
	eDayTo		: E_BA_Weekday		:= E_BA_Weekday.eSunday;
	
	tTime1		: TIME;
	nValue1		: UDINT;
END_VAR

F_BA_SetWeekdays(F_BACnet_SchedWeekly1xM, eDayFrom, eDayTo, 1, tTime1, F_BA_UDIVal(nValue1));

END_FUNCTION

// POUs/Local/Objects/FB_BACnet_Acc
// Accumulator Object
{attribute 'enable_dynamic_creation'}
FUNCTION_BLOCK FB_BACnet_Acc EXTENDS FB_BACnet_BaseAcc
VAR_INPUT
	nVal			: UDINT;	// Process value
	eRlbtyPgm 		: E_BA_Reliability;
END_VAR

SUPER^();

METHOD PROTECTED OnObjectStateChanged
SUPER^.OnObjectStateChanged();

CASE (tState) OF
	TCOM_STATE.TCOM_STATE_PREOP:
		// SyncHandler:
		RequestSyncHandlers(0, 2);
		
		EnableProperty(E_BACnetPropIdentifier.PropValueBeforeChange, FALSE);
		EnableProperty(E_BACnetPropIdentifier.PropValueChangeTime, FALSE);
		EnableProperty(E_BACnetPropIdentifier.PropScale, FALSE);
		EnableProperty(E_BACnetPropIdentifier.PropValueSet, FALSE);
		EnableProperty(E_BACnetPropIdentifier.PropPrescale, FALSE);
		EnableProperty(E_BACnetPropIdentifier.PropLimitMonitoringInverval, FALSE);
		EnableProperty(E_BACnetPropIdentifier.PropPulseRate, FALSE);

	TCOM_STATE.TCOM_STATE_SAFEOP:
		SyncProperty(E_BACnetPropIdentifier.PropPresentValue, SIZEOF(nVal), ADR(nVal), 0, eSync_ToSupplement);
		SyncProperty(E_BACnetPropIdentifier.PropReliability, SIZEOF(eRlbtyPgm), ADR(eRlbtyPgm), 0, eSync_ToSupplement);
			
	TCOM_STATE.TCOM_STATE_OP:
		;
		
END_CASE
END_METHOD

METHOD FB_init : BOOL
VAR_INPUT
	bInitRetains : BOOL; // if TRUE, the retain variables are initialized (warm start / cold start)
	bInCopyCode : BOOL;  // if TRUE, the instance afterwards gets moved into the copy code (online change)
END_VAR
eObjectType := E_BACnetObjType.ObjAccumulator;
END_METHOD

END_FUNCTION_BLOCK

// POUs/Local/Objects/[Base]/FB_BACnet_BaseAcc
// Accumulator Object
{attribute 'enable_dynamic_creation'}
FUNCTION_BLOCK FB_BACnet_BaseAcc EXTENDS FB_BACnet_EventObject
VAR_INPUT CONSTANT PERSISTENT
	{region 'Variable Parameters'}
		{attribute 'parameterCategory':='Value'}
		bOutOfService : BOOL;		
		{attribute 'parameterCategory':='Value'}
		nMaxPresValue : UDINT := 16#FFFFFFFF;
		{attribute 'parameterCategory':='Value'}
			 
		eUnit : E_BA_Unit := E_BA_Unit.eOther_NoUnits; 
		{attribute 'parameterCategory':='Hardware'}
		{attribute 'TcEncoding':='UTF-8'}
		sDeviceType : STRING;	
			 
		{attribute 'parameterCategory':='EventConfig'}
		bLowLimitEnable : BOOL := FALSE;
		{attribute 'parameterCategory':='EventConfig'}
		nLowLimit : UDINT;	
		{attribute 'parameterCategory':='EventConfig'}
		bHighLimitEnable : BOOL := FALSE;
		{attribute 'parameterCategory':='EventConfig'}
		nHighLimit : UDINT;	
	{endregion}	
END_VAR
VAR_OUTPUT
	nPresVal			: UDINT;
END_VAR

SUPER^();

METHOD PROTECTED OnObjectStateChanged
SUPER^.OnObjectStateChanged();

CASE (tState) OF
	TCOM_STATE.TCOM_STATE_PREOP:
		// SyncHandler:
		RequestSyncHandlers(9, 8);
		
	TCOM_STATE.TCOM_STATE_SAFEOP:
		SyncProperty(E_BACnetPropIdentifier.PropPresentValue, SIZEOF(nPresVal), ADR(nPresVal), 0, eSync_FromSupplement);
	
	TCOM_STATE.TCOM_STATE_OP:
		SyncProperty(E_BACnetPropIdentifier.PropOutOfService, SIZEOF(bOutOfService), ADR(bOutOfService), 0, eFullSync_InitPLC);
		SyncProperty(E_BACnetPropIdentifier.PropUnits, SIZEOF(eUnit), ADR(eUnit), 0, eFullSync_InitPLC);
		SyncProperty(E_BACnetPropIdentifier.PropMaxPresValue, SIZEOF(nMaxPresValue), ADR(nMaxPresValue), 0, eFullSync_InitPLC);
	
		SyncProperty(E_BACnetPropIdentifier.PropDeviceType, SIZEOF(sDeviceType), ADR(sDeviceType), 0, eFullSync_InitPLC);
	
		SyncPropertyIdx(E_BACnetPropIdentifier.PropLimitEnable, SIZEOF(BOOL), ADR(bHighLimitEnable), E_BACnet_LimitEnableBits.eHighLimit, 0, eFullSync_InitPLC);	
		SyncPropertyIdx(E_BACnetPropIdentifier.PropLimitEnable, SIZEOF(BOOL), ADR(bLowLimitEnable), E_BACnet_LimitEnableBits.eLowLimit, 0, eFullSync_InitPLC);
		SyncProperty(E_BACnetPropIdentifier.PropHighLimit, SIZEOF(nHighLimit), ADR(nHighLimit), 0, eFullSync_InitPLC);
		SyncProperty(E_BACnetPropIdentifier.PropLowLimit, SIZEOF(nLowLimit), ADR(nLowLimit), 0, eFullSync_InitPLC);
		
END_CASE
END_METHOD

METHOD FB_init : BOOL
VAR_INPUT
	bInitRetains : BOOL; // if TRUE, the retain variables are initialized (warm start / cold start)
	bInCopyCode : BOOL;  // if TRUE, the instance afterwards gets moved into the copy code (online change)
END_VAR
eObjectType := E_BACnetObjType.ObjAccumulator;
END_METHOD

END_FUNCTION_BLOCK

// POUs/Local/Objects/FB_BACnet_PC
// Pulse Converter Object
{attribute 'enable_dynamic_creation'}
FUNCTION_BLOCK FB_BACnet_PC EXTENDS FB_BACnet_EventObject
VAR_INPUT CONSTANT PERSISTENT
	{region 'Variable Parameters'}
		{attribute 'parameterCategory':='Config'}
		stInputReference : ST_BACnet_ObjectPropertyReference;
	{endregion}
END_VAR

SUPER^();

METHOD PROTECTED OnObjectStateChanged
SUPER^.OnObjectStateChanged();

CASE (tState) OF
	TCOM_STATE.TCOM_STATE_PREOP:
		// SyncHandler:
		RequestSyncHandlers(1, 1);
		
	TCOM_STATE.TCOM_STATE_SAFEOP:
		;
	TCOM_STATE.TCOM_STATE_OP:
		// Validate referred property:
		IF (ValidateReference(stInputReference.iObject, stInputReference.tObjectID, 16#FF)) THEN
			InputReference := stInputReference;
		END_IF	
END_CASE
END_METHOD

PROPERTY InputReference : ST_BACnet_ObjectPropertyReference
GET
InputReference := stInputReference;
END_GET
SET
stInputReference := InputReference;

WritePropertyReference(E_BACnetPropIdentifier.PropInputReference, stInputReference);
END_SET
END_PROPERTY

METHOD FB_init : BOOL
VAR_INPUT
	bInitRetains : BOOL; // if TRUE, the retain variables are initialized (warm start / cold start)
	bInCopyCode : BOOL;  // if TRUE, the instance afterwards gets moved into the copy code (online change)
END_VAR
eObjectType := E_BACnetObjType.ObjPulseConverter;
END_METHOD

END_FUNCTION_BLOCK

// POUs/Helper/[internal]/Remote/F_BACnetRM_GetWriteEntrySize
{attribute 'hide'}
FUNCTION F_BACnetRM_GetWriteEntrySize : UDINT
VAR_INPUT
	entry : ST_BACnetRM_WriteEntry;
END_VAR
VAR
END_VAR

IF entry.pNull <> 0 AND_THEN entry.pNull^ THEN
	F_BACnetRM_GetWriteEntrySize:=0;
	RETURN;
END_IF
IF entry.ePropID = E_BACnetPropIdentifier.PropEventEnable OR  entry.ePropID = E_BACnetPropIdentifier.PropLimitEnable THEN
	F_BACnetRM_GetWriteEntrySize:=2;
	RETURN;
END_IF

F_BACnetRM_GetWriteEntrySize:=entry.nData;

END_FUNCTION

// POUs/Helper/[internal]/Remote/F_BACnetRM_IsErrorSet
{attribute 'hide'}
FUNCTION F_BACnetRM_IsErrorSet : BOOL
VAR_INPUT
	stResult	: POINTER TO SendDataRequestResult;
END_VAR
VAR
END_VAR

F_BACnetRM_IsErrorSet:=TRUE;
IF stResult^.errorType = E_BACnet_ErrorType.eAbort AND stResult^.abortReason = E_BACnet_AbortReason.NoReason THEN
	F_BACnetRM_IsErrorSet:=FALSE;
	RETURN;
END_IF
IF stResult^.errorType = E_BACnet_ErrorType.eError AND stResult^.errorClass = E_BACnet_ErrorClass.NoError THEN
	F_BACnetRM_IsErrorSet:=FALSE;
	RETURN;
END_IF
IF stResult^.errorType = E_BACnet_ErrorType.eReject AND stResult^.rejectCode = E_BACnet_RejectReason.NoReason THEN
	F_BACnetRM_IsErrorSet:=FALSE;
	RETURN;
END_IF

END_FUNCTION

// POUs/Helper/[internal]/Remote/F_IsCovProperty
{attribute 'hide'}
FUNCTION F_IsCovProperty : BOOL
VAR_INPUT
	eObjectType			: E_BACnetObjType;
	ePropID				: E_BACnetPropIdentifier;
END_VAR

